LIN {X 0,Y 524.833,Z 335.716,A -85,B 0,C 180,E1 -4782.371,E2 -4782.371} C_VEL
LIN {X 0,Y 525.078,Z 323.315,A -85,B 0,C 180,E1 -4782.955,E2 -4782.955} C_VEL
LIN {X 0,Y 525.315,Z 310.12,A -85,B 0,C 180,E1 -4783.392,E2 -4783.392} C_VEL
LIN {X 0,Y 525.496,Z 297.421,A -85,B 0,C 180,E1 -4783.658,E2 -4783.658} C_VEL
LIN {X 0,Y 525.833,Z 204.394,A -85,B 0,C 180,E1 -4784.955,E2 -4784.955} C_VEL
LIN {X 0,Y 524.222,Z 193.612,A -85,B 0,C 180,E1 -4785.172,E2 -4785.172} C_VEL
LIN {X 0,Y 524.567,Z 175.695,A -85,B 0,C 180,E1 -4787.966,E2 -4787.966} C_VEL
LIN {X 0,Y 525.031,Z 156.558,A -85,B 0,C 180,E1 -4790.981,E2 -4790.981} C_VEL
LIN {X 0,Y 525.12,Z 144.956,A -85,B 0,C 180,E1 -4792.837,E2 -4792.837} C_VEL
LIN {X 0,Y 523.906,Z 138.227,A -85,B 0,C 180,E1 -4794.007,E2 -4794.007} C_VEL
LIN {X 0,Y 523.89,Z 138.23,A -85,B 0,C 180,E1 -4797.136,E2 -4797.136} C_VEL
LIN {X 0,Y 523.864,Z 138.233,A -85,B 0,C 180,E1 -4799.76,E2 -4799.76} C_VEL
LIN {X 0,Y 523.897,Z 138.225,A -85,B 0,C 180,E1 -4802.451,E2 -4802.451} C_VEL
LIN {X 0,Y 523.903,Z 138.229,A -85,B 0,C 180,E1 -4805.227,E2 -4805.227} C_VEL
LIN {X 0,Y 523.895,Z 138.223,A -85,B 0,C 180,E1 -4808.103,E2 -4808.103} C_VEL
LIN {X 0,Y 523.908,Z 138.227,A -85,B 0,C 180,E1 -4811.304,E2 -4811.304} C_VEL
LIN {X 0,Y 523.93,Z 138.224,A -85,B 0,C 180,E1 -4814.688,E2 -4814.688} C_VEL
LIN {X 0,Y 523.886,Z 138.222,A -85,B 0,C 180,E1 -4817.874,E2 -4817.874} C_VEL
LIN {X 0,Y 523.898,Z 138.229,A -85,B 0,C 180,E1 -4820.913,E2 -4820.913} C_VEL
LIN {X 0,Y 523.857,Z 138.225,A -85,B 0,C 180,E1 -4823.821,E2 -4823.821} C_VEL
LIN {X 0,Y 523.906,Z 138.226,A -85,B 0,C 180,E1 -4826.633,E2 -4826.633} C_VEL
LIN {X 0,Y 523.9,Z 138.22,A -85,B 0,C 180,E1 -4829.352,E2 -4829.352} C_VEL
LIN {X 0,Y 523.904,Z 138.225,A -85,B 0,C 180,E1 -4832.295,E2 -4832.295} C_VEL
LIN {X 0,Y 523.894,Z 138.222,A -85,B 0,C 180,E1 -4835.426,E2 -4835.426} C_VEL
LIN {X 0,Y 523.912,Z 138.219,A -85,B 0,C 180,E1 -4837.938,E2 -4837.938} C_VEL
LIN {X 0,Y 523.918,Z 138.225,A -85,B 0,C 180,E1 -4840.405,E2 -4840.405} C_VEL
LIN {X 0,Y 523.911,Z 138.222,A -85,B 0,C 180,E1 -4842.835,E2 -4842.835} C_VEL
LIN {X 0,Y 523.953,Z 138.213,A -85,B 0,C 180,E1 -4845.235,E2 -4845.235} C_VEL
LIN {X 0,Y 523.951,Z 138.22,A -85,B 0,C 180,E1 -4848.392,E2 -4848.392} C_VEL
LIN {X 0,Y 523.937,Z 138.217,A -85,B 0,C 180,E1 -4851.515,E2 -4851.515} C_VEL
LIN {X 0,Y 524.02,Z 138.206,A -85,B 0,C 180,E1 -4854.613,E2 -4854.613} C_VEL
LIN {X 0,Y 524.096,Z 138.202,A -85,B 0,C 180,E1 -4857.694,E2 -4857.694} C_VEL
LIN {X 0,Y 524.088,Z 138.205,A -85,B 0,C 180,E1 -4860,E2 -4860} C_VEL
LIN {X 0,Y 524.095,Z 138.2,A -85,B 0,C 180,E1 -4862.305,E2 -4862.305} C_VEL
LIN {X 0,Y 523.992,Z 138.214,A -85,B 0,C 180,E1 -4866.159,E2 -4866.159} C_VEL
LIN {X 0,Y 523.936,Z 138.221,A -85,B 0,C 180,E1 -4869.263,E2 -4869.263} C_VEL
LIN {X 0,Y 523.936,Z 138.22,A -85,B 0,C 180,E1 -4872.393,E2 -4872.393} C_VEL
LIN {X 0,Y 523.901,Z 138.231,A -85,B 0,C 180,E1 -4875.562,E2 -4875.562} C_VEL
LIN {X 0,Y 523.915,Z 138.221,A -85,B 0,C 180,E1 -4878.78,E2 -4878.78} C_VEL
LIN {X 0,Y 523.913,Z 138.227,A -85,B 0,C 180,E1 -4881.234,E2 -4881.234} C_VEL
LIN {X 0,Y 523.955,Z 138.316,A -85,B 0,C 180,E1 -4883.702,E2 -4883.702} C_VEL
LIN {X 0,Y 524.545,Z 142.807,A -85,B 0,C 180,E1 -4884.541,E2 -4884.541} C_VEL
LIN {X 0,Y 524.355,Z 157.183,A -85,B 0,C 180,E1 -4887.11,E2 -4887.11} C_VEL
LIN {X 0,Y 524.273,Z 167.066,A -85,B 0,C 180,E1 -4888.896,E2 -4888.896} C_VEL
LIN {X 0,Y 526.014,Z 177.203,A -85,B 0,C 180,E1 -4889.102,E2 -4889.102} C_VEL
LIN {X 0,Y 525.462,Z 274.648,A -85,B 0,C 180,E1 -4890.477,E2 -4890.477} C_VEL
LIN {X 0,Y 525.278,Z 287.649,A -85,B 0,C 180,E1 -4890.817,E2 -4890.817} C_VEL
LIN {X 0,Y 525.102,Z 299.989,A -85,B 0,C 180,E1 -4891.293,E2 -4891.293} C_VEL
LIN {X 0,Y 524.906,Z 309.383,A -85,B 0,C 180,E1 -4891.77,E2 -4891.77} C_VEL
LIN {X 0,Y 524.16,Z 314.614,A -85,B 0,C 180,E1 -4892.061,E2 -4892.061} C_VEL
LIN {X 0,Y 521.076,Z 322.898,A -85,B 0,C 180,E1 -4892.559,E2 -4892.559} C_VEL
LIN {X 0,Y 517.989,Z 330.723,A -85,B 0,C 180,E1 -4893.137,E2 -4893.137} C_VEL
LIN {X 0,Y 517.24,Z 335.226,A -85,B 0,C 180,E1 -4893.55,E2 -4893.55} C_VEL
LIN {X 0,Y 516.94,Z 344.855,A -85,B 0,C 180,E1 -4894.603,E2 -4894.603} C_VEL
LIN {X 0,Y 516.707,Z 353.618,A -85,B 0,C 180,E1 -4895.793,E2 -4895.793} C_VEL
LIN {X 0,Y 516.51,Z 360.825,A -85,B 0,C 180,E1 -4897.02,E2 -4897.02} C_VEL
LIN {X 0,Y 516.44,Z 366.704,A -85,B 0,C 180,E1 -4898.29,E2 -4898.29} C_VEL
LIN {X 0,Y 516.325,Z 370.782,A -85,B 0,C 180,E1 -4899.42,E2 -4899.42} C_VEL
LIN {X 0,Y 516.282,Z 374.444,A -85,B 0,C 180,E1 -4900.799,E2 -4900.799} C_VEL
LIN {X 0,Y 516.213,Z 376.306,A -85,B 0,C 180,E1 -4901.844,E2 -4901.844} C_VEL
LIN {X 0,Y 516.185,Z 377.467,A -85,B 0,C 180,E1 -4902.903,E2 -4902.903} C_VEL
LIN {X 0,Y 516.194,Z 377.886,A -85,B 0,C 180,E1 -4903.976,E2 -4903.976} C_VEL
LIN {X 0,Y 516.243,Z 377.53,A -85,B 0,C 180,E1 -4905.065,E2 -4905.065} C_VEL
LIN {X 0,Y 516.199,Z 376.374,A -85,B 0,C 180,E1 -4906.185,E2 -4906.185} C_VEL
LIN {X 0,Y 516.272,Z 373.361,A -85,B 0,C 180,E1 -4907.745,E2 -4907.745} C_VEL
LIN {X 0,Y 516.343,Z 370.205,A -85,B 0,C 180,E1 -4908.84,E2 -4908.84} C_VEL
LIN {X 0,Y 516.438,Z 364.785,A -85,B 0,C 180,E1 -4910.239,E2 -4910.239} C_VEL
LIN {X 0,Y 516.611,Z 358.52,A -85,B 0,C 180,E1 -4911.483,E2 -4911.483} C_VEL
LIN {X 0,Y 516.789,Z 350.403,A -85,B 0,C 180,E1 -4912.76,E2 -4912.76} C_VEL
LIN {X 0,Y 517.042,Z 341.469,A -85,B 0,C 180,E1 -4913.873,E2 -4913.873} C_VEL
LIN {X 0,Y 517.345,Z 331.353,A -85,B 0,C 180,E1 -4914.895,E2 -4914.895} C_VEL
LIN {X 0,Y 517.662,Z 320.358,A -85,B 0,C 180,E1 -4915.787,E2 -4915.787} C_VEL
LIN {X 0,Y 517.936,Z 308.363,A -85,B 0,C 180,E1 -4916.548,E2 -4916.548} C_VEL
LIN {X 0,Y 518.223,Z 297.272,A -85,B 0,C 180,E1 -4917.091,E2 -4917.091} C_VEL
LIN {X 0,Y 518.402,Z 284.135,A -85,B 0,C 180,E1 -4917.565,E2 -4917.565} C_VEL
LIN {X 0,Y 518.581,Z 270.861,A -85,B 0,C 180,E1 -4917.865,E2 -4917.865} C_VEL
LIN {X 0,Y 519.017,Z 176.794,A -85,B 0,C 180,E1 -4919.202,E2 -4919.202} C_VEL
LIN {X 0,Y 517.248,Z 167.254,A -85,B 0,C 180,E1 -4919.397,E2 -4919.397} C_VEL
LIN {X 0,Y 517.574,Z 152.214,A -85,B 0,C 180,E1 -4922.24,E2 -4922.24} C_VEL
LIN {X 0,Y 517.649,Z 143.381,A -85,B 0,C 180,E1 -4923.934,E2 -4923.934} C_VEL
LIN {X 0,Y 516.888,Z 139.103,A -85,B 0,C 180,E1 -4924.802,E2 -4924.802} C_VEL
LIN {X 0,Y 516.865,Z 139.099,A -85,B 0,C 180,E1 -4927.622,E2 -4927.622} C_VEL
LIN {X 0,Y 516.909,Z 139.096,A -85,B 0,C 180,E1 -4930.129,E2 -4930.129} C_VEL
LIN {X 0,Y 516.874,Z 139.103,A -85,B 0,C 180,E1 -4932.595,E2 -4932.595} C_VEL
LIN {X 0,Y 516.928,Z 139.091,A -85,B 0,C 180,E1 -4935.03,E2 -4935.03} C_VEL
LIN {X 0,Y 516.921,Z 139.097,A -85,B 0,C 180,E1 -4938.233,E2 -4938.233} C_VEL
LIN {X 0,Y 516.915,Z 139.091,A -85,B 0,C 180,E1 -4941.399,E2 -4941.399} C_VEL
LIN {X 0,Y 516.976,Z 139.087,A -85,B 0,C 180,E1 -4944.54,E2 -4944.54} C_VEL
LIN {X 0,Y 517.069,Z 139.074,A -85,B 0,C 180,E1 -4947.663,E2 -4947.663} C_VEL
LIN {X 0,Y 517.061,Z 139.08,A -85,B 0,C 180,E1 -4950,E2 -4950} C_VEL
LIN {X 0,Y 517.069,Z 139.076,A -85,B 0,C 180,E1 -4952.337,E2 -4952.337} C_VEL
LIN {X 0,Y 516.964,Z 139.089,A -85,B 0,C 180,E1 -4956.244,E2 -4956.244} C_VEL
LIN {X 0,Y 516.903,Z 139.095,A -85,B 0,C 180,E1 -4959.39,E2 -4959.39} C_VEL
LIN {X 0,Y 516.893,Z 139.094,A -85,B 0,C 180,E1 -4962.565,E2 -4962.565} C_VEL
LIN {X 0,Y 516.932,Z 139.09,A -85,B 0,C 180,E1 -4965.142,E2 -4965.142} C_VEL
LIN {X 0,Y 516.865,Z 139.099,A -85,B 0,C 180,E1 -4968.224,E2 -4968.224} C_VEL
LIN {X 0,Y 516.866,Z 139.097,A -85,B 0,C 180,E1 -4970.703,E2 -4970.703} C_VEL
LIN {X 0,Y 516.835,Z 139.105,A -85,B 0,C 180,E1 -4973.225,E2 -4973.225} C_VEL
LIN {X 0,Y 516.874,Z 139.097,A -85,B 0,C 180,E1 -4976.181,E2 -4976.181} C_VEL
LIN {X 0,Y 516.824,Z 139.102,A -85,B 0,C 180,E1 -4978.421,E2 -4978.421} C_VEL
LIN {X 0,Y 516.872,Z 139.101,A -85,B 0,C 180,E1 -4981.11,E2 -4981.11} C_VEL
LIN {X 0,Y 516.875,Z 139.097,A -85,B 0,C 180,E1 -4983.961,E2 -4983.961} C_VEL
LIN {X 0,Y 516.843,Z 139.102,A -85,B 0,C 180,E1 -4986.748,E2 -4986.748} C_VEL
LIN {X 0,Y 516.852,Z 139.101,A -85,B 0,C 180,E1 -4989.724,E2 -4989.724} C_VEL
LIN {X 0,Y 516.835,Z 139.105,A -85,B 0,C 180,E1 -4992.836,E2 -4992.836} C_VEL
LIN {X 0,Y 516.89,Z 139.102,A -85,B 0,C 180,E1 -4995.007,E2 -4995.007} C_VEL
LIN {X 0,Y 516.846,Z 139.101,A -85,B 0,C 180,E1 -4998.406,E2 -4998.406} C_VEL
LIN {X 0,Y 516.866,Z 139.101,A -85,B 0,C 180,E1 -5001.283,E2 -5001.283} C_VEL
LIN {X 0,Y 516.844,Z 139.106,A -85,B 0,C 180,E1 -5004.673,E2 -5004.673} C_VEL
LIN {X 0,Y 516.885,Z 139.096,A -85,B 0,C 180,E1 -5007.458,E2 -5007.458} C_VEL
LIN {X 0,Y 516.89,Z 139.103,A -85,B 0,C 180,E1 -5010.694,E2 -5010.694} C_VEL
LIN {X 0,Y 516.872,Z 139.096,A -85,B 0,C 180,E1 -5013.819,E2 -5013.819} C_VEL
LIN {X 0,Y 516.834,Z 139.107,A -85,B 0,C 180,E1 -5016.775,E2 -5016.775} C_VEL
LIN {X 0,Y 516.899,Z 139.093,A -85,B 0,C 180,E1 -5019.742,E2 -5019.742} C_VEL
LIN {X 0,Y 516.871,Z 139.103,A -85,B 0,C 180,E1 -5022.595,E2 -5022.595} C_VEL
LIN {X 0,Y 516.925,Z 139.091,A -85,B 0,C 180,E1 -5025.03,E2 -5025.03} C_VEL
LIN {X 0,Y 516.918,Z 139.098,A -85,B 0,C 180,E1 -5028.233,E2 -5028.233} C_VEL
LIN {X 0,Y 516.912,Z 139.091,A -85,B 0,C 180,E1 -5031.399,E2 -5031.399} C_VEL
LIN {X 0,Y 516.973,Z 139.087,A -85,B 0,C 180,E1 -5034.54,E2 -5034.54} C_VEL
LIN {X 0,Y 517.066,Z 139.075,A -85,B 0,C 180,E1 -5037.663,E2 -5037.663} C_VEL
LIN {X 0,Y 517.058,Z 139.081,A -85,B 0,C 180,E1 -5040,E2 -5040} C_VEL
LIN {X 0,Y 517.066,Z 139.076,A -85,B 0,C 180,E1 -5042.337,E2 -5042.337} C_VEL
LIN {X 0,Y 516.961,Z 139.089,A -85,B 0,C 180,E1 -5046.244,E2 -5046.244} C_VEL
LIN {X 0,Y 516.9,Z 139.095,A -85,B 0,C 180,E1 -5049.391,E2 -5049.391} C_VEL
LIN {X 0,Y 516.89,Z 139.094,A -85,B 0,C 180,E1 -5052.565,E2 -5052.565} C_VEL
LIN {X 0,Y 516.93,Z 139.091,A -85,B 0,C 180,E1 -5055.142,E2 -5055.142} C_VEL
LIN {X 0,Y 516.864,Z 139.099,A -85,B 0,C 180,E1 -5058.225,E2 -5058.225} C_VEL
LIN {X 0,Y 516.865,Z 139.097,A -85,B 0,C 180,E1 -5060.704,E2 -5060.704} C_VEL
LIN {X 0,Y 516.834,Z 139.105,A -85,B 0,C 180,E1 -5063.226,E2 -5063.226} C_VEL
LIN {X 0,Y 516.874,Z 139.097,A -85,B 0,C 180,E1 -5066.182,E2 -5066.182} C_VEL
LIN {X 0,Y 516.824,Z 139.102,A -85,B 0,C 180,E1 -5068.421,E2 -5068.421} C_VEL
LIN {X 0,Y 516.844,Z 139.105,A -85,B 0,C 180,E1 -5071.113,E2 -5071.113} C_VEL
LIN {X 0,Y 516.876,Z 139.097,A -85,B 0,C 180,E1 -5073.962,E2 -5073.962} C_VEL
LIN {X 0,Y 516.811,Z 139.106,A -85,B 0,C 180,E1 -5076.752,E2 -5076.752} C_VEL
LIN {X 0,Y 516.853,Z 139.1,A -85,B 0,C 180,E1 -5079.724,E2 -5079.724} C_VEL
LIN {X 0,Y 516.838,Z 139.105,A -85,B 0,C 180,E1 -5082.837,E2 -5082.837} C_VEL
LIN {X 0,Y 516.894,Z 139.102,A -85,B 0,C 180,E1 -5085.007,E2 -5085.007} C_VEL
LIN {X 0,Y 516.847,Z 139.101,A -85,B 0,C 180,E1 -5088.408,E2 -5088.408} C_VEL
LIN {X 0,Y 516.867,Z 139.1,A -85,B 0,C 180,E1 -5091.283,E2 -5091.283} C_VEL
LIN {X 0,Y 516.847,Z 139.106,A -85,B 0,C 180,E1 -5094.674,E2 -5094.674} C_VEL
LIN {X 0,Y 516.866,Z 139.098,A -85,B 0,C 180,E1 -5097.462,E2 -5097.462} C_VEL
LIN {X 0,Y 516.837,Z 139.107,A -85,B 0,C 180,E1 -5100.491,E2 -5100.491} C_VEL
LIN {X 0,Y 516.828,Z 139.103,A -85,B 0,C 180,E1 -5103.337,E2 -5103.337} C_VEL
LIN {X 0,Y 516.857,Z 139.147,A -85,B 0,C 180,E1 -5105.691,E2 -5105.691} C_VEL
LIN {X 0,Y 518.326,Z 147.13,A -85,B 0,C 180,E1 -5107.091,E2 -5107.091} C_VEL
LIN {X 0,Y 518.015,Z 161.935,A -85,B 0,C 180,E1 -5109.52,E2 -5109.52} C_VEL
LIN {X 0,Y 517.575,Z 178.892,A -85,B 0,C 180,E1 -5112.257,E2 -5112.257} C_VEL
LIN {X 0,Y 517.266,Z 193.985,A -85,B 0,C 180,E1 -5114.641,E2 -5114.641} C_VEL
LIN {X 0,Y 519.025,Z 206.11,A -85,B 0,C 180,E1 -5114.869,E2 -5114.869} C_VEL
LIN {X 0,Y 518.545,Z 302.791,A -85,B 0,C 180,E1 -5116.255,E2 -5116.255} C_VEL
LIN {X 0,Y 518.28,Z 316.493,A -85,B 0,C 180,E1 -5116.622,E2 -5116.622} C_VEL
LIN {X 0,Y 518.045,Z 328.834,A -85,B 0,C 180,E1 -5117.115,E2 -5117.115} C_VEL
LIN {X 0,Y 517.691,Z 341.583,A -85,B 0,C 180,E1 -5117.81,E2 -5117.81} C_VEL
LIN {X 0,Y 517.429,Z 353.383,A -85,B 0,C 180,E1 -5118.642,E2 -5118.642} C_VEL
LIN {X 0,Y 517.158,Z 362.386,A -85,B 0,C 180,E1 -5119.429,E2 -5119.429} C_VEL
LIN {X 0,Y 516.9,Z 371.625,A -85,B 0,C 180,E1 -5120.412,E2 -5120.412} C_VEL
LIN {X 0,Y 516.652,Z 380.613,A -85,B 0,C 180,E1 -5121.591,E2 -5121.591} C_VEL
LIN {X 0,Y 516.503,Z 387.85,A -85,B 0,C 180,E1 -5122.769,E2 -5122.769} C_VEL
LIN {X 0,Y 516.385,Z 392.73,A -85,B 0,C 180,E1 -5123.749,E2 -5123.749} C_VEL
LIN {X 0,Y 516.312,Z 397.472,A -85,B 0,C 180,E1 -5124.924,E2 -5124.924} C_VEL
LIN {X 0,Y 516.352,Z 401.097,A -85,B 0,C 180,E1 -5126.098,E2 -5126.098} C_VEL
LIN {X 0,Y 516.283,Z 402.964,A -85,B 0,C 180,E1 -5126.879,E2 -5126.879} C_VEL
LIN {X 0,Y 516.261,Z 404.365,A -85,B 0,C 180,E1 -5127.659,E2 -5127.659} C_VEL
LIN {X 0,Y 516.162,Z 405.968,A -85,B 0,C 180,E1 -5129.22,E2 -5129.22} C_VEL
LIN {X 0,Y 516.159,Z 406.183,A -85,B 0,C 180,E1 -5130,E2 -5130} C_VEL
LIN {X 0,Y 516.192,Z 405.353,A -85,B 0,C 180,E1 -5131.56,E2 -5131.56} C_VEL
LIN {X 0,Y 516.261,Z 404.351,A -85,B 0,C 180,E1 -5132.34,E2 -5132.34} C_VEL
LIN {X 0,Y 516.282,Z 402.945,A -85,B 0,C 180,E1 -5133.121,E2 -5133.121} C_VEL
LIN {X 0,Y 516.31,Z 399.992,A -85,B 0,C 180,E1 -5134.293,E2 -5134.293} C_VEL
LIN {X 0,Y 516.368,Z 395.995,A -85,B 0,C 180,E1 -5135.467,E2 -5135.467} C_VEL
LIN {X 0,Y 516.44,Z 390.084,A -85,B 0,C 180,E1 -5136.792,E2 -5136.792} C_VEL
LIN {X 0,Y 516.586,Z 383.121,A -85,B 0,C 180,E1 -5138.016,E2 -5138.016} C_VEL
LIN {X 0,Y 516.772,Z 374.778,A -85,B 0,C 180,E1 -5139.195,E2 -5139.195} C_VEL
LIN {X 0,Y 516.997,Z 366.207,A -85,B 0,C 180,E1 -5140.179,E2 -5140.179} C_VEL
LIN {X 0,Y 517.317,Z 355.623,A -85,B 0,C 180,E1 -5141.162,E2 -5141.162} C_VEL
LIN {X 0,Y 517.608,Z 344.508,A -85,B 0,C 180,E1 -5141.994,E2 -5141.994} C_VEL
LIN {X 0,Y 517.939,Z 333.614,A -85,B 0,C 180,E1 -5142.638,E2 -5142.638} C_VEL
LIN {X 0,Y 518.168,Z 321.669,A -85,B 0,C 180,E1 -5143.181,E2 -5143.181} C_VEL
LIN {X 0,Y 518.445,Z 307.88,A -85,B 0,C 180,E1 -5143.623,E2 -5143.623} C_VEL
LIN {X 0,Y 518.626,Z 295.308,A -85,B 0,C 180,E1 -5143.868,E2 -5143.868} C_VEL
LIN {X 0,Y 518.957,Z 204.938,A -85,B 0,C 180,E1 -5145.147,E2 -5145.147} C_VEL
LIN {X 0,Y 517.222,Z 193.364,A -85,B 0,C 180,E1 -5145.387,E2 -5145.387} C_VEL
LIN {X 0,Y 517.665,Z 174.314,A -85,B 0,C 180,E1 -5148.4,E2 -5148.4} C_VEL
LIN {X 0,Y 518.083,Z 155.034,A -85,B 0,C 180,E1 -5151.485,E2 -5151.485} C_VEL
LIN {X 0,Y 518.193,Z 146.314,A -85,B 0,C 180,E1 -5152.899,E2 -5152.899} C_VEL
LIN {X 0,Y 516.869,Z 139.103,A -85,B 0,C 180,E1 -5154.169,E2 -5154.169} C_VEL
LIN {X 0,Y 516.827,Z 139.107,A -85,B 0,C 180,E1 -5156.663,E2 -5156.663} C_VEL
LIN {X 0,Y 516.836,Z 139.112,A -85,B 0,C 180,E1 -5159.508,E2 -5159.508} C_VEL
LIN {X 0,Y 516.865,Z 139.101,A -85,B 0,C 180,E1 -5162.537,E2 -5162.537} C_VEL
LIN {X 0,Y 516.846,Z 139.108,A -85,B 0,C 180,E1 -5165.326,E2 -5165.326} C_VEL
LIN {X 0,Y 516.865,Z 139.103,A -85,B 0,C 180,E1 -5168.716,E2 -5168.716} C_VEL
LIN {X 0,Y 516.841,Z 139.103,A -85,B 0,C 180,E1 -5171.781,E2 -5171.781} C_VEL
LIN {X 0,Y 516.892,Z 139.102,A -85,B 0,C 180,E1 -5175.006,E2 -5175.006} C_VEL
LIN {X 0,Y 516.843,Z 139.102,A -85,B 0,C 180,E1 -5178.406,E2 -5178.406} C_VEL
LIN {X 0,Y 516.864,Z 139.101,A -85,B 0,C 180,E1 -5181.282,E2 -5181.282} C_VEL
LIN {X 0,Y 516.845,Z 139.107,A -85,B 0,C 180,E1 -5184.672,E2 -5184.672} C_VEL
LIN {X 0,Y 516.886,Z 139.095,A -85,B 0,C 180,E1 -5187.457,E2 -5187.457} C_VEL
LIN {X 0,Y 516.819,Z 139.11,A -85,B 0,C 180,E1 -5190.689,E2 -5190.689} C_VEL
LIN {X 0,Y 516.83,Z 139.1,A -85,B 0,C 180,E1 -5193.337,E2 -5193.337} C_VEL
LIN {X 0,Y 516.873,Z 139.098,A -85,B 0,C 180,E1 -5195.926,E2 -5195.926} C_VEL
LIN {X 0,Y 516.845,Z 139.107,A -85,B 0,C 180,E1 -5198.46,E2 -5198.46} C_VEL
LIN {X 0,Y 516.856,Z 139.098,A -85,B 0,C 180,E1 -5200.953,E2 -5200.953} C_VEL
LIN {X 0,Y 516.832,Z 139.102,A -85,B 0,C 180,E1 -5203.407,E2 -5203.407} C_VEL
LIN {X 0,Y 516.861,Z 139.099,A -85,B 0,C 180,E1 -5205.832,E2 -5205.832} C_VEL
LIN {X 0,Y 516.917,Z 139.097,A -85,B 0,C 180,E1 -5208.232,E2 -5208.232} C_VEL
LIN {X 0,Y 516.911,Z 139.092,A -85,B 0,C 180,E1 -5211.398,E2 -5211.398} C_VEL
LIN {X 0,Y 516.971,Z 139.085,A -85,B 0,C 180,E1 -5214.539,E2 -5214.539} C_VEL
LIN {X 0,Y 517.065,Z 139.077,A -85,B 0,C 180,E1 -5217.663,E2 -5217.663} C_VEL
LIN {X 0,Y 517.056,Z 139.081,A -85,B 0,C 180,E1 -5220,E2 -5220} C_VEL
LIN {X 0,Y 517.064,Z 139.076,A -85,B 0,C 180,E1 -5222.337,E2 -5222.337} C_VEL
LIN {X 0,Y 516.959,Z 139.09,A -85,B 0,C 180,E1 -5226.243,E2 -5226.243} C_VEL
LIN {X 0,Y 516.898,Z 139.099,A -85,B 0,C 180,E1 -5229.39,E2 -5229.39} C_VEL
LIN {X 0,Y 516.888,Z 139.098,A -85,B 0,C 180,E1 -5232.565,E2 -5232.565} C_VEL
LIN {X 0,Y 516.927,Z 139.096,A -85,B 0,C 180,E1 -5235.142,E2 -5235.142} C_VEL
LIN {X 0,Y 516.864,Z 139.1,A -85,B 0,C 180,E1 -5238.224,E2 -5238.224} C_VEL
LIN {X 0,Y 516.881,Z 139.099,A -85,B 0,C 180,E1 -5240.702,E2 -5240.702} C_VEL
LIN {X 0,Y 516.916,Z 139.208,A -85,B 0,C 180,E1 -5243.566,E2 -5243.566} C_VEL
LIN {X 0,Y 517.58,Z 144.348,A -85,B 0,C 180,E1 -5244.529,E2 -5244.529} C_VEL
LIN {X 0,Y 517.381,Z 159.561,A -85,B 0,C 180,E1 -5247.287,E2 -5247.287} C_VEL
LIN {X 0,Y 517.289,Z 167.305,A -85,B 0,C 180,E1 -5248.697,E2 -5248.697} C_VEL
LIN {X 0,Y 519.071,Z 177.126,A -85,B 0,C 180,E1 -5248.894,E2 -5248.894} C_VEL
LIN {X 0,Y 518.568,Z 275.171,A -85,B 0,C 180,E1 -5250.306,E2 -5250.306} C_VEL
LIN {X 0,Y 518.367,Z 288.716,A -85,B 0,C 180,E1 -5250.671,E2 -5250.671} C_VEL
LIN {X 0,Y 518.18,Z 299.936,A -85,B 0,C 180,E1 -5251.114,E2 -5251.114} C_VEL
LIN {X 0,Y 517.874,Z 312.383,A -85,B 0,C 180,E1 -5251.772,E2 -5251.772} C_VEL
LIN {X 0,Y 517.567,Z 324.128,A -85,B 0,C 180,E1 -5252.582,E2 -5252.582} C_VEL
LIN {X 0,Y 517.245,Z 334.754,A -85,B 0,C 180,E1 -5253.503,E2 -5253.503} C_VEL
LIN {X 0,Y 517.24,Z 335.226,A -85,B 0,C 180,E1 -5253.55,E2 -5253.55} C_VEL
LIN {X 0,Y 516.498,Z 339.613,A -85,B 0,C 180,E1 -5253.989,E2 -5253.989} C_VEL
LIN {X 0,Y 513.417,Z 346.426,A -85,B 0,C 180,E1 -5254.721,E2 -5254.721} C_VEL
LIN {X 0,Y 510.347,Z 352.625,A -85,B 0,C 180,E1 -5255.514,E2 -5255.514} C_VEL
LIN {X 0,Y 509.621,Z 356.065,A -85,B 0,C 180,E1 -5256.042,E2 -5256.042} C_VEL
LIN {X 0,Y 509.438,Z 363.245,A -85,B 0,C 180,E1 -5257.373,E2 -5257.373} C_VEL
LIN {X 0,Y 509.344,Z 367.586,A -85,B 0,C 180,E1 -5258.383,E2 -5258.383} C_VEL
LIN {X 0,Y 509.223,Z 372.606,A -85,B 0,C 180,E1 -5259.923,E2 -5259.923} C_VEL
LIN {X 0,Y 509.196,Z 374.321,A -85,B 0,C 180,E1 -5260.615,E2 -5260.615} C_VEL
LIN {X 0,Y 509.117,Z 376.485,A -85,B 0,C 180,E1 -5261.805,E2 -5261.805} C_VEL
LIN {X 0,Y 509.097,Z 377.713,A -85,B 0,C 180,E1 -5262.976,E2 -5262.976} C_VEL
LIN {X 0,Y 509.11,Z 378.078,A -85,B 0,C 180,E1 -5264.125,E2 -5264.125} C_VEL
LIN {X 0,Y 509.142,Z 377.615,A -85,B 0,C 180,E1 -5265.253,E2 -5265.253} C_VEL
LIN {X 0,Y 509.108,Z 376.365,A -85,B 0,C 180,E1 -5266.353,E2 -5266.353} C_VEL
LIN {X 0,Y 509.145,Z 374.368,A -85,B 0,C 180,E1 -5267.44,E2 -5267.44} C_VEL
LIN {X 0,Y 509.272,Z 370.168,A -85,B 0,C 180,E1 -5268.975,E2 -5268.975} C_VEL
LIN {X 0,Y 509.371,Z 364.864,A -85,B 0,C 180,E1 -5270.349,E2 -5270.349} C_VEL
LIN {X 0,Y 509.569,Z 358.394,A -85,B 0,C 180,E1 -5271.638,E2 -5271.638} C_VEL
LIN {X 0,Y 509.757,Z 350.41,A -85,B 0,C 180,E1 -5272.902,E2 -5272.902} C_VEL
LIN {X 0,Y 510.045,Z 341.308,A -85,B 0,C 180,E1 -5274.045,E2 -5274.045} C_VEL
LIN {X 0,Y 510.341,Z 331.71,A -85,B 0,C 180,E1 -5275.025,E2 -5275.025} C_VEL
LIN {X 0,Y 510.674,Z 321.298,A -85,B 0,C 180,E1 -5275.889,E2 -5275.889} C_VEL
LIN {X 0,Y 510.99,Z 309.187,A -85,B 0,C 180,E1 -5276.678,E2 -5276.678} C_VEL
LIN {X 0,Y 511.308,Z 296.926,A -85,B 0,C 180,E1 -5277.289,E2 -5277.289} C_VEL
LIN {X 0,Y 511.518,Z 283.934,A -85,B 0,C 180,E1 -5277.756,E2 -5277.756} C_VEL
LIN {X 0,Y 511.714,Z 270.642,A -85,B 0,C 180,E1 -5278.056,E2 -5278.056} C_VEL
LIN {X 0,Y 512.281,Z 178.46,A -85,B 0,C 180,E1 -5279.382,E2 -5279.382} C_VEL
LIN {X 0,Y 510.264,Z 167.381,A -85,B 0,C 180,E1 -5279.617,E2 -5279.617} C_VEL
LIN {X 0,Y 510.608,Z 152.103,A -85,B 0,C 180,E1 -5282.543,E2 -5282.543} C_VEL
LIN {X 0,Y 510.729,Z 145.206,A -85,B 0,C 180,E1 -5283.875,E2 -5283.875} C_VEL
LIN {X 0,Y 509.845,Z 139.98,A -85,B 0,C 180,E1 -5284.974,E2 -5284.974} C_VEL
LIN {X 0,Y 509.804,Z 139.982,A -85,B 0,C 180,E1 -5288.148,E2 -5288.148} C_VEL
LIN {X 0,Y 509.839,Z 139.98,A -85,B 0,C 180,E1 -5290.681,E2 -5290.681} C_VEL
LIN {X 0,Y 509.791,Z 139.979,A -85,B 0,C 180,E1 -5293.172,E2 -5293.172} C_VEL
LIN {X 0,Y 509.84,Z 139.973,A -85,B 0,C 180,E1 -5295.634,E2 -5295.634} C_VEL
LIN {X 0,Y 509.885,Z 139.972,A -85,B 0,C 180,E1 -5298.131,E2 -5298.131} C_VEL
LIN {X 0,Y 509.868,Z 139.969,A -85,B 0,C 180,E1 -5301.279,E2 -5301.279} C_VEL
LIN {X 0,Y 509.912,Z 139.965,A -85,B 0,C 180,E1 -5303.67,E2 -5303.67} C_VEL
LIN {X 0,Y 509.881,Z 139.968,A -85,B 0,C 180,E1 -5306.84,E2 -5306.84} C_VEL
LIN {X 0,Y 509.919,Z 139.967,A -85,B 0,C 180,E1 -5308.421,E2 -5308.421} C_VEL
LIN {X 0,Y 510.03,Z 139.956,A -85,B 0,C 180,E1 -5310,E2 -5310} C_VEL
LIN {X 0,Y 510.038,Z 139.952,A -85,B 0,C 180,E1 -5312.369,E2 -5312.369} C_VEL
LIN {X 0,Y 509.931,Z 139.964,A -85,B 0,C 180,E1 -5315.536,E2 -5315.536} C_VEL
LIN {X 0,Y 509.871,Z 139.977,A -85,B 0,C 180,E1 -5317.923,E2 -5317.923} C_VEL
LIN {X 0,Y 509.858,Z 139.971,A -85,B 0,C 180,E1 -5321.127,E2 -5321.127} C_VEL
LIN {X 0,Y 509.82,Z 139.98,A -85,B 0,C 180,E1 -5323.553,E2 -5323.553} C_VEL
LIN {X 0,Y 509.798,Z 139.982,A -85,B 0,C 180,E1 -5326.005,E2 -5326.005} C_VEL
LIN {X 0,Y 509.822,Z 139.975,A -85,B 0,C 180,E1 -5328.485,E2 -5328.485} C_VEL
LIN {X 0,Y 509.813,Z 139.977,A -85,B 0,C 180,E1 -5331.003,E2 -5331.003} C_VEL
LIN {X 0,Y 509.803,Z 139.986,A -85,B 0,C 180,E1 -5333.565,E2 -5333.565} C_VEL
LIN {X 0,Y 509.81,Z 139.976,A -85,B 0,C 180,E1 -5336.356,E2 -5336.356} C_VEL
LIN {X 0,Y 509.788,Z 139.98,A -85,B 0,C 180,E1 -5338.849,E2 -5338.849} C_VEL
LIN {X 0,Y 509.806,Z 139.982,A -85,B 0,C 180,E1 -5341.591,E2 -5341.591} C_VEL
LIN {X 0,Y 509.828,Z 139.974,A -85,B 0,C 180,E1 -5344.415,E2 -5344.415} C_VEL
LIN {X 0,Y 509.8,Z 139.985,A -85,B 0,C 180,E1 -5347.342,E2 -5347.342} C_VEL
LIN {X 0,Y 509.806,Z 139.977,A -85,B 0,C 180,E1 -5350.385,E2 -5350.385} C_VEL
LIN {X 0,Y 509.799,Z 139.98,A -85,B 0,C 180,E1 -5353.573,E2 -5353.573} C_VEL
LIN {X 0,Y 509.799,Z 139.979,A -85,B 0,C 180,E1 -5356.426,E2 -5356.426} C_VEL
LIN {X 0,Y 509.807,Z 139.977,A -85,B 0,C 180,E1 -5359.615,E2 -5359.615} C_VEL
LIN {X 0,Y 509.776,Z 139.985,A -85,B 0,C 180,E1 -5362.656,E2 -5362.656} C_VEL
LIN {X 0,Y 509.831,Z 139.973,A -85,B 0,C 180,E1 -5365.801,E2 -5365.801} C_VEL
LIN {X 0,Y 509.83,Z 139.982,A -85,B 0,C 180,E1 -5368.722,E2 -5368.722} C_VEL
LIN {X 0,Y 509.823,Z 139.977,A -85,B 0,C 180,E1 -5371.153,E2 -5371.153} C_VEL
LIN {X 0,Y 509.84,Z 139.972,A -85,B 0,C 180,E1 -5373.826,E2 -5373.826} C_VEL
LIN {X 0,Y 509.801,Z 139.983,A -85,B 0,C 180,E1 -5376.436,E2 -5376.436} C_VEL
LIN {X 0,Y 509.882,Z 139.968,A -85,B 0,C 180,E1 -5379.844,E2 -5379.844} C_VEL
LIN {X 0,Y 509.845,Z 139.979,A -85,B 0,C 180,E1 -5382.347,E2 -5382.347} C_VEL
LIN {X 0,Y 509.877,Z 139.971,A -85,B 0,C 180,E1 -5384.818,E2 -5384.818} C_VEL
LIN {X 0,Y 509.882,Z 139.973,A -85,B 0,C 180,E1 -5388.131,E2 -5388.131} C_VEL
LIN {X 0,Y 509.865,Z 139.969,A -85,B 0,C 180,E1 -5391.279,E2 -5391.279} C_VEL
LIN {X 0,Y 509.909,Z 139.965,A -85,B 0,C 180,E1 -5393.67,E2 -5393.67} C_VEL
LIN {X 0,Y 509.878,Z 139.968,A -85,B 0,C 180,E1 -5396.84,E2 -5396.84} C_VEL
LIN {X 0,Y 509.916,Z 139.967,A -85,B 0,C 180,E1 -5398.421,E2 -5398.421} C_VEL
LIN {X 0,Y 510.027,Z 139.957,A -85,B 0,C 180,E1 -5400,E2 -5400} C_VEL
LIN {X 0,Y 510.035,Z 139.952,A -85,B 0,C 180,E1 -5402.37,E2 -5402.37} C_VEL
LIN {X 0,Y 509.928,Z 139.964,A -85,B 0,C 180,E1 -5405.537,E2 -5405.537} C_VEL
LIN {X 0,Y 509.868,Z 139.977,A -85,B 0,C 180,E1 -5407.923,E2 -5407.923} C_VEL
LIN {X 0,Y 509.856,Z 139.971,A -85,B 0,C 180,E1 -5411.127,E2 -5411.127} C_VEL
LIN {X 0,Y 509.817,Z 139.981,A -85,B 0,C 180,E1 -5413.554,E2 -5413.554} C_VEL
LIN {X 0,Y 509.796,Z 139.982,A -85,B 0,C 180,E1 -5416.005,E2 -5416.005} C_VEL
LIN {X 0,Y 509.82,Z 139.975,A -85,B 0,C 180,E1 -5418.486,E2 -5418.486} C_VEL
LIN {X 0,Y 509.812,Z 139.977,A -85,B 0,C 180,E1 -5421.004,E2 -5421.004} C_VEL
LIN {X 0,Y 509.802,Z 139.985,A -85,B 0,C 180,E1 -5423.565,E2 -5423.565} C_VEL
LIN {X 0,Y 509.81,Z 139.976,A -85,B 0,C 180,E1 -5426.357,E2 -5426.357} C_VEL
LIN {X 0,Y 509.788,Z 139.98,A -85,B 0,C 180,E1 -5428.85,E2 -5428.85} C_VEL
LIN {X 0,Y 509.792,Z 139.983,A -85,B 0,C 180,E1 -5431.592,E2 -5431.592} C_VEL
LIN {X 0,Y 509.829,Z 139.974,A -85,B 0,C 180,E1 -5434.416,E2 -5434.416} C_VEL
LIN {X 0,Y 509.779,Z 139.987,A -85,B 0,C 180,E1 -5437.344,E2 -5437.344} C_VEL
LIN {X 0,Y 509.809,Z 139.976,A -85,B 0,C 180,E1 -5440.385,E2 -5440.385} C_VEL
LIN {X 0,Y 509.79,Z 139.981,A -85,B 0,C 180,E1 -5443.575,E2 -5443.575} C_VEL
LIN {X 0,Y 509.79,Z 139.98,A -85,B 0,C 180,E1 -5446.426,E2 -5446.426} C_VEL
LIN {X 0,Y 509.81,Z 139.977,A -85,B 0,C 180,E1 -5449.616,E2 -5449.616} C_VEL
LIN {X 0,Y 509.778,Z 139.985,A -85,B 0,C 180,E1 -5452.656,E2 -5452.656} C_VEL
LIN {X 0,Y 509.837,Z 139.972,A -85,B 0,C 180,E1 -5455.801,E2 -5455.801} C_VEL
LIN {X 0,Y 509.814,Z 139.984,A -85,B 0,C 180,E1 -5458.727,E2 -5458.727} C_VEL
LIN {X 0,Y 509.822,Z 139.977,A -85,B 0,C 180,E1 -5462.051,E2 -5462.051} C_VEL
LIN {X 0,Y 509.783,Z 139.984,A -85,B 0,C 180,E1 -5464.699,E2 -5464.699} C_VEL
LIN {X 0,Y 509.824,Z 140.059,A -85,B 0,C 180,E1 -5465.52,E2 -5465.52} C_VEL
LIN {X 0,Y 511.39,Z 148.609,A -85,B 0,C 180,E1 -5467.041,E2 -5467.041} C_VEL
LIN {X 0,Y 511.01,Z 163.768,A -85,B 0,C 180,E1 -5469.56,E2 -5469.56} C_VEL
LIN {X 0,Y 510.593,Z 179.025,A -85,B 0,C 180,E1 -5472.058,E2 -5472.058} C_VEL
LIN {X 0,Y 510.228,Z 193.618,A -85,B 0,C 180,E1 -5474.421,E2 -5474.421} C_VEL
LIN {X 0,Y 512.206,Z 207.217,A -85,B 0,C 180,E1 -5474.681,E2 -5474.681} C_VEL
LIN {X 0,Y 511.649,Z 302.381,A -85,B 0,C 180,E1 -5476.066,E2 -5476.066} C_VEL
LIN {X 0,Y 511.385,Z 316.153,A -85,B 0,C 180,E1 -5476.438,E2 -5476.438} C_VEL
LIN {X 0,Y 511.084,Z 328.539,A -85,B 0,C 180,E1 -5476.936,E2 -5476.936} C_VEL
LIN {X 0,Y 510.743,Z 341.132,A -85,B 0,C 180,E1 -5477.63,E2 -5477.63} C_VEL
LIN {X 0,Y 510.484,Z 351.842,A -85,B 0,C 180,E1 -5478.384,E2 -5478.384} C_VEL
LIN {X 0,Y 510.161,Z 362.147,A -85,B 0,C 180,E1 -5479.282,E2 -5479.282} C_VEL
LIN {X 0,Y 509.847,Z 371.396,A -85,B 0,C 180,E1 -5480.278,E2 -5480.278} C_VEL
LIN {X 0,Y 509.606,Z 380.394,A -85,B 0,C 180,E1 -5481.474,E2 -5481.474} C_VEL
LIN {X 0,Y 509.428,Z 387.637,A -85,B 0,C 180,E1 -5482.668,E2 -5482.668} C_VEL
LIN {X 0,Y 509.309,Z 392.523,A -85,B 0,C 180,E1 -5483.662,E2 -5483.662} C_VEL
LIN {X 0,Y 509.241,Z 397.271,A -85,B 0,C 180,E1 -5484.853,E2 -5484.853} C_VEL
LIN {X 0,Y 509.245,Z 400.899,A -85,B 0,C 180,E1 -5486.043,E2 -5486.043} C_VEL
LIN {X 0,Y 509.2,Z 402.769,A -85,B 0,C 180,E1 -5486.835,E2 -5486.835} C_VEL
LIN {X 0,Y 509.19,Z 404.17,A -85,B 0,C 180,E1 -5487.627,E2 -5487.627} C_VEL
LIN {X 0,Y 509.076,Z 405.774,A -85,B 0,C 180,E1 -5489.209,E2 -5489.209} C_VEL
LIN {X 0,Y 509.07,Z 405.989,A -85,B 0,C 180,E1 -5490,E2 -5490} C_VEL
LIN {X 0,Y 509.113,Z 405.156,A -85,B 0,C 180,E1 -5491.582,E2 -5491.582} C_VEL
LIN {X 0,Y 509.19,Z 404.153,A -85,B 0,C 180,E1 -5492.373,E2 -5492.373} C_VEL
LIN {X 0,Y 509.2,Z 402.744,A -85,B 0,C 180,E1 -5493.165,E2 -5493.165} C_VEL
LIN {X 0,Y 509.202,Z 399.786,A -85,B 0,C 180,E1 -5494.353,E2 -5494.353} C_VEL
LIN {X 0,Y 509.283,Z 395.783,A -85,B 0,C 180,E1 -5495.543,E2 -5495.543} C_VEL
LIN {X 0,Y 509.395,Z 389.723,A -85,B 0,C 180,E1 -5496.914,E2 -5496.914} C_VEL
LIN {X 0,Y 509.536,Z 382.889,A -85,B 0,C 180,E1 -5498.127,E2 -5498.127} C_VEL
LIN {X 0,Y 509.732,Z 374.535,A -85,B 0,C 180,E1 -5499.323,E2 -5499.323} C_VEL
LIN {X 0,Y 509.969,Z 365.95,A -85,B 0,C 180,E1 -5500.32,E2 -5500.32} C_VEL
LIN {X 0,Y 510.333,Z 355.35,A -85,B 0,C 180,E1 -5501.317,E2 -5501.317} C_VEL
LIN {X 0,Y 510.644,Z 344.218,A -85,B 0,C 180,E1 -5502.16,E2 -5502.16} C_VEL
LIN {X 0,Y 510.989,Z 333.296,A -85,B 0,C 180,E1 -5502.813,E2 -5502.813} C_VEL
LIN {X 0,Y 511.246,Z 321.315,A -85,B 0,C 180,E1 -5503.363,E2 -5503.363} C_VEL
LIN {X 0,Y 511.559,Z 307.477,A -85,B 0,C 180,E1 -5503.81,E2 -5503.81} C_VEL
LIN {X 0,Y 511.736,Z 294.745,A -85,B 0,C 180,E1 -5504.058,E2 -5504.058} C_VEL
LIN {X 0,Y 512.136,Z 205.897,A -85,B 0,C 180,E1 -5505.336,E2 -5505.336} C_VEL
LIN {X 0,Y 510.213,Z 193.274,A -85,B 0,C 180,E1 -5505.586,E2 -5505.586} C_VEL
LIN {X 0,Y 510.679,Z 174.096,A -85,B 0,C 180,E1 -5508.661,E2 -5508.661} C_VEL
LIN {X 0,Y 511.131,Z 156.099,A -85,B 0,C 180,E1 -5511.58,E2 -5511.58} C_VEL
LIN {X 0,Y 511.279,Z 147.899,A -85,B 0,C 180,E1 -5512.93,E2 -5512.93} C_VEL
LIN {X 0,Y 509.816,Z 139.981,A -85,B 0,C 180,E1 -5514.32,E2 -5514.32} C_VEL
LIN {X 0,Y 509.813,Z 139.983,A -85,B 0,C 180,E1 -5517.059,E2 -5517.059} C_VEL
LIN {X 0,Y 509.782,Z 139.988,A -85,B 0,C 180,E1 -5519.755,E2 -5519.755} C_VEL
LIN {X 0,Y 509.824,Z 139.98,A -85,B 0,C 180,E1 -5522.765,E2 -5522.765} C_VEL
LIN {X 0,Y 509.791,Z 139.983,A -85,B 0,C 180,E1 -5525.572,E2 -5525.572} C_VEL
LIN {X 0,Y 509.81,Z 139.979,A -85,B 0,C 180,E1 -5528.341,E2 -5528.341} C_VEL
LIN {X 0,Y 509.798,Z 139.983,A -85,B 0,C 180,E1 -5531.43,E2 -5531.43} C_VEL
LIN {X 0,Y 509.836,Z 139.98,A -85,B 0,C 180,E1 -5534.669,E2 -5534.669} C_VEL
LIN {X 0,Y 509.783,Z 139.98,A -85,B 0,C 180,E1 -5537.505,E2 -5537.505} C_VEL
LIN {X 0,Y 509.822,Z 139.98,A -85,B 0,C 180,E1 -5540.645,E2 -5540.645} C_VEL
LIN {X 0,Y 509.766,Z 139.98,A -85,B 0,C 180,E1 -5543.642,E2 -5543.642} C_VEL
LIN {X 0,Y 509.832,Z 139.979,A -85,B 0,C 180,E1 -5546.537,E2 -5546.537} C_VEL
LIN {X 0,Y 509.795,Z 139.977,A -85,B 0,C 180,E1 -5549.331,E2 -5549.331} C_VEL
LIN {X 0,Y 509.815,Z 139.978,A -85,B 0,C 180,E1 -5552.05,E2 -5552.05} C_VEL
LIN {X 0,Y 509.793,Z 139.985,A -85,B 0,C 180,E1 -5554.699,E2 -5554.699} C_VEL
LIN {X 0,Y 509.817,Z 139.972,A -85,B 0,C 180,E1 -5557.458,E2 -5557.458} C_VEL
LIN {X 0,Y 509.817,Z 139.978,A -85,B 0,C 180,E1 -5560.679,E2 -5560.679} C_VEL
LIN {X 0,Y 509.787,Z 139.98,A -85,B 0,C 180,E1 -5563.171,E2 -5563.171} C_VEL
LIN {X 0,Y 509.835,Z 139.973,A -85,B 0,C 180,E1 -5565.633,E2 -5565.633} C_VEL
LIN {X 0,Y 509.881,Z 139.973,A -85,B 0,C 180,E1 -5568.13,E2 -5568.13} C_VEL
LIN {X 0,Y 509.864,Z 139.969,A -85,B 0,C 180,E1 -5571.279,E2 -5571.279} C_VEL
LIN {X 0,Y 509.907,Z 139.968,A -85,B 0,C 180,E1 -5573.669,E2 -5573.669} C_VEL
LIN {X 0,Y 509.875,Z 139.969,A -85,B 0,C 180,E1 -5576.839,E2 -5576.839} C_VEL
LIN {X 0,Y 509.913,Z 139.967,A -85,B 0,C 180,E1 -5578.42,E2 -5578.42} C_VEL
LIN {X 0,Y 510.025,Z 139.957,A -85,B 0,C 180,E1 -5580,E2 -5580} C_VEL
LIN {X 0,Y 510.033,Z 139.951,A -85,B 0,C 180,E1 -5582.369,E2 -5582.369} C_VEL
LIN {X 0,Y 509.927,Z 139.967,A -85,B 0,C 180,E1 -5585.536,E2 -5585.536} C_VEL
LIN {X 0,Y 509.865,Z 139.978,A -85,B 0,C 180,E1 -5587.923,E2 -5587.923} C_VEL
LIN {X 0,Y 509.853,Z 139.975,A -85,B 0,C 180,E1 -5591.126,E2 -5591.126} C_VEL
LIN {X 0,Y 509.831,Z 139.984,A -85,B 0,C 180,E1 -5593.553,E2 -5593.553} C_VEL
LIN {X 0,Y 509.79,Z 139.985,A -85,B 0,C 180,E1 -5596.005,E2 -5596.005} C_VEL
LIN {X 0,Y 509.823,Z 139.977,A -85,B 0,C 180,E1 -5598.485,E2 -5598.485} C_VEL
LIN {X 0,Y 509.823,Z 139.981,A -85,B 0,C 180,E1 -5601.002,E2 -5601.002} C_VEL
LIN {X 0,Y 509.847,Z 140.109,A -85,B 0,C 180,E1 -5603.428,E2 -5603.428} C_VEL
LIN {X 0,Y 510.594,Z 145.126,A -85,B 0,C 180,E1 -5604.389,E2 -5604.389} C_VEL
LIN {X 0,Y 510.393,Z 160.754,A -85,B 0,C 180,E1 -5607.248,E2 -5607.248} C_VEL
LIN {X 0,Y 510.323,Z 167.43,A -85,B 0,C 180,E1 -5608.473,E2 -5608.473} C_VEL
LIN {X 0,Y 512.244,Z 178.077,A -85,B 0,C 180,E1 -5608.698,E2 -5608.698} C_VEL
LIN {X 0,Y 511.688,Z 274.684,A -85,B 0,C 180,E1 -5610.107,E2 -5610.107} C_VEL
LIN {X 0,Y 511.478,Z 288.021,A -85,B 0,C 180,E1 -5610.463,E2 -5610.463} C_VEL
LIN {X 0,Y 511.262,Z 300.832,A -85,B 0,C 180,E1 -5610.972,E2 -5610.972} C_VEL
LIN {X 0,Y 510.925,Z 312.919,A -85,B 0,C 180,E1 -5611.629,E2 -5611.629} C_VEL
LIN {X 0,Y 510.576,Z 324.832,A -85,B 0,C 180,E1 -5612.468,E2 -5612.468} C_VEL
LIN {X 0,Y 510.278,Z 334.037,A -85,B 0,C 180,E1 -5613.274,E2 -5613.274} C_VEL
LIN {X 0,Y 510.014,Z 343.03,A -85,B 0,C 180,E1 -5614.23,E2 -5614.23} C_VEL
LIN {X 0,Y 509.762,Z 351.809,A -85,B 0,C 180,E1 -5615.383,E2 -5615.383} C_VEL
LIN {X 0,Y 509.621,Z 356.065,A -85,B 0,C 180,E1 -5616.042,E2 -5616.042} C_VEL
LIN {X 0,Y 508.924,Z 359.349,A -85,B 0,C 180,E1 -5616.589,E2 -5616.589} C_VEL
LIN {X 0,Y 505.952,Z 364.267,A -85,B 0,C 180,E1 -5617.504,E2 -5617.504} C_VEL
LIN {X 0,Y 502.937,Z 368.439,A -85,B 0,C 180,E1 -5618.472,E2 -5618.472} C_VEL
LIN {X 0,Y 502.185,Z 370.558,A -85,B 0,C 180,E1 -5619.097,E2 -5619.097} C_VEL
LIN {X 0,Y 502.141,Z 373.364,A -85,B 0,C 180,E1 -5620.077,E2 -5620.077} C_VEL
LIN {X 0,Y 502.066,Z 375.656,A -85,B 0,C 180,E1 -5621.14,E2 -5621.14} C_VEL
LIN {X 0,Y 501.999,Z 377.255,A -85,B 0,C 180,E1 -5622.221,E2 -5622.221} C_VEL
LIN {X 0,Y 501.992,Z 378.115,A -85,B 0,C 180,E1 -5623.315,E2 -5623.315} C_VEL
LIN {X 0,Y 502.032,Z 378.206,A -85,B 0,C 180,E1 -5624.443,E2 -5624.443} C_VEL
LIN {X 0,Y 502.034,Z 377.523,A -85,B 0,C 180,E1 -5625.578,E2 -5625.578} C_VEL
LIN {X 0,Y 502.031,Z 376.046,A -85,B 0,C 180,E1 -5626.715,E2 -5626.715} C_VEL
LIN {X 0,Y 502.097,Z 373.644,A -85,B 0,C 180,E1 -5627.889,E2 -5627.889} C_VEL
LIN {X 0,Y 502.204,Z 370.218,A -85,B 0,C 180,E1 -5629.085,E2 -5629.085} C_VEL
LIN {X 0,Y 502.289,Z 365.59,A -85,B 0,C 180,E1 -5630.313,E2 -5630.313} C_VEL
LIN {X 0,Y 502.499,Z 359.603,A -85,B 0,C 180,E1 -5631.556,E2 -5631.556} C_VEL
LIN {X 0,Y 502.695,Z 351.862,A -85,B 0,C 180,E1 -5632.834,E2 -5632.834} C_VEL
LIN {X 0,Y 502.952,Z 343.568,A -85,B 0,C 180,E1 -5633.941,E2 -5633.941} C_VEL
LIN {X 0,Y 503.34,Z 334.192,A -85,B 0,C 180,E1 -5634.956,E2 -5634.956} C_VEL
LIN {X 0,Y 503.646,Z 323.944,A -85,B 0,C 180,E1 -5635.856,E2 -5635.856} C_VEL
LIN {X 0,Y 503.981,Z 312.45,A -85,B 0,C 180,E1 -5636.665,E2 -5636.665} C_VEL
LIN {X 0,Y 504.329,Z 300.451,A -85,B 0,C 180,E1 -5637.317,E2 -5637.317} C_VEL
LIN {X 0,Y 504.578,Z 286.916,A -85,B 0,C 180,E1 -5637.852,E2 -5637.852} C_VEL
LIN {X 0,Y 504.779,Z 274.261,A -85,B 0,C 180,E1 -5638.185,E2 -5638.185} C_VEL
LIN {X 0,Y 505.326,Z 178.628,A -85,B 0,C 180,E1 -5639.595,E2 -5639.595} C_VEL
LIN {X 0,Y 503.295,Z 167.518,A -85,B 0,C 180,E1 -5639.84,E2 -5639.84} C_VEL
LIN {X 0,Y 503.712,Z 151.438,A -85,B 0,C 180,E1 -5642.954,E2 -5642.954} C_VEL
LIN {X 0,Y 503.753,Z 146.458,A -85,B 0,C 180,E1 -5643.931,E2 -5643.931} C_VEL
LIN {X 0,Y 502.775,Z 140.86,A -85,B 0,C 180,E1 -5645.096,E2 -5645.096} C_VEL
LIN {X 0,Y 502.768,Z 140.856,A -85,B 0,C 180,E1 -5647.826,E2 -5647.826} C_VEL
LIN {X 0,Y 502.798,Z 140.857,A -85,B 0,C 180,E1 -5650.4,E2 -5650.4} C_VEL
LIN {X 0,Y 502.752,Z 140.858,A -85,B 0,C 180,E1 -5652.929,E2 -5652.929} C_VEL
LIN {X 0,Y 502.821,Z 140.846,A -85,B 0,C 180,E1 -5655.429,E2 -5655.429} C_VEL
LIN {X 0,Y 502.833,Z 140.849,A -85,B 0,C 180,E1 -5658.716,E2 -5658.716} C_VEL
LIN {X 0,Y 502.842,Z 140.848,A -85,B 0,C 180,E1 -5661.966,E2 -5661.966} C_VEL
LIN {X 0,Y 502.888,Z 140.844,A -85,B 0,C 180,E1 -5664.386,E2 -5664.386} C_VEL
LIN {X 0,Y 503.005,Z 140.825,A -85,B 0,C 180,E1 -5667.598,E2 -5667.598} C_VEL
LIN {X 0,Y 502.999,Z 140.832,A -85,B 0,C 180,E1 -5670,E2 -5670} C_VEL
LIN {X 0,Y 503.005,Z 140.827,A -85,B 0,C 180,E1 -5672.402,E2 -5672.402} C_VEL
LIN {X 0,Y 502.888,Z 140.842,A -85,B 0,C 180,E1 -5675.614,E2 -5675.614} C_VEL
LIN {X 0,Y 502.842,Z 140.851,A -85,B 0,C 180,E1 -5678.034,E2 -5678.034} C_VEL
LIN {X 0,Y 502.833,Z 140.847,A -85,B 0,C 180,E1 -5681.284,E2 -5681.284} C_VEL
LIN {X 0,Y 502.82,Z 140.847,A -85,B 0,C 180,E1 -5684.571,E2 -5684.571} C_VEL
LIN {X 0,Y 502.779,Z 140.857,A -85,B 0,C 180,E1 -5687.91,E2 -5687.91} C_VEL
LIN {X 0,Y 502.798,Z 140.849,A -85,B 0,C 180,E1 -5690.528,E2 -5690.528} C_VEL
LIN {X 0,Y 502.777,Z 140.854,A -85,B 0,C 180,E1 -5693.041,E2 -5693.041} C_VEL
LIN {X 0,Y 502.772,Z 140.859,A -85,B 0,C 180,E1 -5695.679,E2 -5695.679} C_VEL
LIN {X 0,Y 502.754,Z 140.855,A -85,B 0,C 180,E1 -5698.378,E2 -5698.378} C_VEL
LIN {X 0,Y 502.78,Z 140.859,A -85,B 0,C 180,E1 -5701.497,E2 -5701.497} C_VEL
LIN {X 0,Y 502.78,Z 140.852,A -85,B 0,C 180,E1 -5704.441,E2 -5704.441} C_VEL
LIN {X 0,Y 502.756,Z 140.862,A -85,B 0,C 180,E1 -5707.175,E2 -5707.175} C_VEL
LIN {X 0,Y 502.764,Z 140.854,A -85,B 0,C 180,E1 -5710.017,E2 -5710.017} C_VEL
LIN {X 0,Y 502.74,Z 140.864,A -85,B 0,C 180,E1 -5713.234,E2 -5713.234} C_VEL
LIN {X 0,Y 502.772,Z 140.854,A -85,B 0,C 180,E1 -5715.66,E2 -5715.66} C_VEL
LIN {X 0,Y 502.758,Z 140.863,A -85,B 0,C 180,E1 -5719.012,E2 -5719.012} C_VEL
LIN {X 0,Y 502.754,Z 140.855,A -85,B 0,C 180,E1 -5722.043,E2 -5722.043} C_VEL
LIN {X 0,Y 502.776,Z 140.858,A -85,B 0,C 180,E1 -5725.033,E2 -5725.033} C_VEL
LIN {X 0,Y 502.771,Z 140.853,A -85,B 0,C 180,E1 -5727.915,E2 -5727.915} C_VEL
LIN {X 0,Y 502.782,Z 140.86,A -85,B 0,C 180,E1 -5730.71,E2 -5730.71} C_VEL
LIN {X 0,Y 502.766,Z 140.854,A -85,B 0,C 180,E1 -5733.46,E2 -5733.46} C_VEL
LIN {X 0,Y 502.753,Z 140.857,A -85,B 0,C 180,E1 -5736.085,E2 -5736.085} C_VEL
LIN {X 0,Y 502.762,Z 140.861,A -85,B 0,C 180,E1 -5738.688,E2 -5738.688} C_VEL
LIN {X 0,Y 502.798,Z 140.85,A -85,B 0,C 180,E1 -5741.247,E2 -5741.247} C_VEL
LIN {X 0,Y 502.828,Z 140.851,A -85,B 0,C 180,E1 -5744.665,E2 -5744.665} C_VEL
LIN {X 0,Y 502.863,Z 140.846,A -85,B 0,C 180,E1 -5748.044,E2 -5748.044} C_VEL
LIN {X 0,Y 502.829,Z 140.846,A -85,B 0,C 180,E1 -5751.156,E2 -5751.156} C_VEL
LIN {X 0,Y 502.86,Z 140.843,A -85,B 0,C 180,E1 -5753.581,E2 -5753.581} C_VEL
LIN {X 0,Y 502.823,Z 140.847,A -85,B 0,C 180,E1 -5756.795,E2 -5756.795} C_VEL
LIN {X 0,Y 502.886,Z 140.843,A -85,B 0,C 180,E1 -5758.399,E2 -5758.399} C_VEL
LIN {X 0,Y 502.996,Z 140.833,A -85,B 0,C 180,E1 -5760,E2 -5760} C_VEL
LIN {X 0,Y 503.002,Z 140.827,A -85,B 0,C 180,E1 -5762.403,E2 -5762.403} C_VEL
LIN {X 0,Y 502.885,Z 140.843,A -85,B 0,C 180,E1 -5765.614,E2 -5765.614} C_VEL
LIN {X 0,Y 502.84,Z 140.851,A -85,B 0,C 180,E1 -5768.035,E2 -5768.035} C_VEL
LIN {X 0,Y 502.831,Z 140.847,A -85,B 0,C 180,E1 -5771.285,E2 -5771.285} C_VEL
LIN {X 0,Y 502.818,Z 140.847,A -85,B 0,C 180,E1 -5774.572,E2 -5774.572} C_VEL
LIN {X 0,Y 502.778,Z 140.857,A -85,B 0,C 180,E1 -5777.91,E2 -5777.91} C_VEL
LIN {X 0,Y 502.797,Z 140.849,A -85,B 0,C 180,E1 -5780.528,E2 -5780.528} C_VEL
LIN {X 0,Y 502.776,Z 140.854,A -85,B 0,C 180,E1 -5783.042,E2 -5783.042} C_VEL
LIN {X 0,Y 502.771,Z 140.859,A -85,B 0,C 180,E1 -5785.68,E2 -5785.68} C_VEL
LIN {X 0,Y 502.755,Z 140.855,A -85,B 0,C 180,E1 -5788.378,E2 -5788.378} C_VEL
LIN {X 0,Y 502.766,Z 140.86,A -85,B 0,C 180,E1 -5791.495,E2 -5791.495} C_VEL
LIN {X 0,Y 502.781,Z 140.852,A -85,B 0,C 180,E1 -5794.441,E2 -5794.441} C_VEL
LIN {X 0,Y 502.733,Z 140.866,A -85,B 0,C 180,E1 -5797.172,E2 -5797.172} C_VEL
LIN {X 0,Y 502.765,Z 140.854,A -85,B 0,C 180,E1 -5800.018,E2 -5800.018} C_VEL
LIN {X 0,Y 502.737,Z 140.864,A -85,B 0,C 180,E1 -5803.236,E2 -5803.236} C_VEL
LIN {X 0,Y 502.765,Z 140.855,A -85,B 0,C 180,E1 -5805.659,E2 -5805.659} C_VEL
LIN {X 0,Y 502.761,Z 140.862,A -85,B 0,C 180,E1 -5809.013,E2 -5809.013} C_VEL
LIN {X 0,Y 502.757,Z 140.855,A -85,B 0,C 180,E1 -5812.043,E2 -5812.043} C_VEL
LIN {X 0,Y 502.78,Z 140.857,A -85,B 0,C 180,E1 -5815.033,E2 -5815.033} C_VEL
LIN {X 0,Y 502.757,Z 140.855,A -85,B 0,C 180,E1 -5817.914,E2 -5817.914} C_VEL
LIN {X 0,Y 502.752,Z 140.863,A -85,B 0,C 180,E1 -5820.708,E2 -5820.708} C_VEL
LIN {X 0,Y 502.77,Z 140.853,A -85,B 0,C 180,E1 -5823.461,E2 -5823.461} C_VEL
LIN {X 0,Y 502.791,Z 140.982,A -85,B 0,C 180,E1 -5825.348,E2 -5825.348} C_VEL
LIN {X 0,Y 504.451,Z 150.374,A -85,B 0,C 180,E1 -5827.04,E2 -5827.04} C_VEL
LIN {X 0,Y 504.092,Z 163.98,A -85,B 0,C 180,E1 -5829.332,E2 -5829.332} C_VEL
LIN {X 0,Y 503.605,Z 179.585,A -85,B 0,C 180,E1 -5831.924,E2 -5831.924} C_VEL
LIN {X 0,Y 503.256,Z 193.443,A -85,B 0,C 180,E1 -5834.201,E2 -5834.201} C_VEL
LIN {X 0,Y 505.32,Z 208.164,A -85,B 0,C 180,E1 -5834.487,E2 -5834.487} C_VEL
LIN {X 0,Y 504.766,Z 301.941,A -85,B 0,C 180,E1 -5835.872,E2 -5835.872} C_VEL
LIN {X 0,Y 504.483,Z 315.793,A -85,B 0,C 180,E1 -5836.249,E2 -5836.249} C_VEL
LIN {X 0,Y 504.142,Z 328.233,A -85,B 0,C 180,E1 -5836.753,E2 -5836.753} C_VEL
LIN {X 0,Y 503.762,Z 340.912,A -85,B 0,C 180,E1 -5837.459,E2 -5837.459} C_VEL
LIN {X 0,Y 503.471,Z 352.879,A -85,B 0,C 180,E1 -5838.322,E2 -5838.322} C_VEL
LIN {X 0,Y 503.169,Z 361.908,A -85,B 0,C 180,E1 -5839.131,E2 -5839.131} C_VEL
LIN {X 0,Y 502.813,Z 371.169,A -85,B 0,C 180,E1 -5840.141,E2 -5840.141} C_VEL
LIN {X 0,Y 502.554,Z 380.174,A -85,B 0,C 180,E1 -5841.354,E2 -5841.354} C_VEL
LIN {X 0,Y 502.344,Z 387.425,A -85,B 0,C 180,E1 -5842.564,E2 -5842.564} C_VEL
LIN {X 0,Y 502.236,Z 392.317,A -85,B 0,C 180,E1 -5843.572,E2 -5843.572} C_VEL
LIN {X 0,Y 502.172,Z 397.07,A -85,B 0,C 180,E1 -5844.781,E2 -5844.781} C_VEL
LIN {X 0,Y 502.137,Z 400.7,A -85,B 0,C 180,E1 -5845.987,E2 -5845.987} C_VEL
LIN {X 0,Y 502.12,Z 402.573,A -85,B 0,C 180,E1 -5846.79,E2 -5846.79} C_VEL
LIN {X 0,Y 502.092,Z 403.976,A -85,B 0,C 180,E1 -5847.593,E2 -5847.593} C_VEL
LIN {X 0,Y 501.993,Z 405.58,A -85,B 0,C 180,E1 -5849.198,E2 -5849.198} C_VEL
LIN {X 0,Y 501.984,Z 405.795,A -85,B 0,C 180,E1 -5850,E2 -5850} C_VEL
LIN {X 0,Y 502.036,Z 404.959,A -85,B 0,C 180,E1 -5851.604,E2 -5851.604} C_VEL
LIN {X 0,Y 502.092,Z 403.954,A -85,B 0,C 180,E1 -5852.407,E2 -5852.407} C_VEL
LIN {X 0,Y 502.12,Z 402.543,A -85,B 0,C 180,E1 -5853.209,E2 -5853.209} C_VEL
LIN {X 0,Y 502.1,Z 399.579,A -85,B 0,C 180,E1 -5854.415,E2 -5854.415} C_VEL
LIN {X 0,Y 502.199,Z 395.57,A -85,B 0,C 180,E1 -5855.622,E2 -5855.622} C_VEL
LIN {X 0,Y 502.327,Z 389.5,A -85,B 0,C 180,E1 -5857.011,E2 -5857.011} C_VEL
LIN {X 0,Y 502.47,Z 382.657,A -85,B 0,C 180,E1 -5858.242,E2 -5858.242} C_VEL
LIN {X 0,Y 502.706,Z 374.295,A -85,B 0,C 180,E1 -5859.454,E2 -5859.454} C_VEL
LIN {X 0,Y 502.958,Z 365.697,A -85,B 0,C 180,E1 -5860.466,E2 -5860.466} C_VEL
LIN {X 0,Y 503.347,Z 355.086,A -85,B 0,C 180,E1 -5861.476,E2 -5861.476} C_VEL
LIN {X 0,Y 503.658,Z 343.939,A -85,B 0,C 180,E1 -5862.331,E2 -5862.331} C_VEL
LIN {X 0,Y 504.041,Z 332.994,A -85,B 0,C 180,E1 -5862.993,E2 -5862.993} C_VEL
LIN {X 0,Y 504.309,Z 320.979,A -85,B 0,C 180,E1 -5863.55,E2 -5863.55} C_VEL
LIN {X 0,Y 504.645,Z 308.01,A -85,B 0,C 180,E1 -5863.977,E2 -5863.977} C_VEL
LIN {X 0,Y 504.847,Z 294.224,A -85,B 0,C 180,E1 -5864.254,E2 -5864.254} C_VEL
LIN {X 0,Y 505.32,Z 206.973,A -85,B 0,C 180,E1 -5865.53,E2 -5865.53} C_VEL
LIN {X 0,Y 503.204,Z 193.012,A -85,B 0,C 180,E1 -5865.817,E2 -5865.817} C_VEL
LIN {X 0,Y 503.731,Z 173.876,A -85,B 0,C 180,E1 -5868.928,E2 -5868.928} C_VEL
LIN {X 0,Y 504.18,Z 157.185,A -85,B 0,C 180,E1 -5871.678,E2 -5871.678} C_VEL
LIN {X 0,Y 504.259,Z 148.723,A -85,B 0,C 180,E1 -5873.094,E2 -5873.094} C_VEL
LIN {X 0,Y 502.769,Z 140.86,A -85,B 0,C 180,E1 -5874.505,E2 -5874.505} C_VEL
LIN {X 0,Y 502.767,Z 140.865,A -85,B 0,C 180,E1 -5877.47,E2 -5877.47} C_VEL
LIN {X 0,Y 502.741,Z 140.863,A -85,B 0,C 180,E1 -5880.215,E2 -5880.215} C_VEL
LIN {X 0,Y 502.797,Z 140.858,A -85,B 0,C 180,E1 -5883.033,E2 -5883.033} C_VEL
LIN {X 0,Y 502.742,Z 140.859,A -85,B 0,C 180,E1 -5885.953,E2 -5885.953} C_VEL
LIN {X 0,Y 502.777,Z 140.861,A -85,B 0,C 180,E1 -5888.977,E2 -5888.977} C_VEL
LIN {X 0,Y 502.741,Z 140.86,A -85,B 0,C 180,E1 -5892.191,E2 -5892.191} C_VEL
LIN {X 0,Y 502.774,Z 140.856,A -85,B 0,C 180,E1 -5895.47,E2 -5895.47} C_VEL
LIN {X 0,Y 502.756,Z 140.863,A -85,B 0,C 180,E1 -5898.927,E2 -5898.927} C_VEL
LIN {X 0,Y 502.755,Z 140.856,A -85,B 0,C 180,E1 -5902.042,E2 -5902.042} C_VEL
LIN {X 0,Y 502.777,Z 140.857,A -85,B 0,C 180,E1 -5905.032,E2 -5905.032} C_VEL
LIN {X 0,Y 502.766,Z 140.854,A -85,B 0,C 180,E1 -5907.914,E2 -5907.914} C_VEL
LIN {X 0,Y 502.745,Z 140.862,A -85,B 0,C 180,E1 -5910.707,E2 -5910.707} C_VEL
LIN {X 0,Y 502.767,Z 140.851,A -85,B 0,C 180,E1 -5913.459,E2 -5913.459} C_VEL
LIN {X 0,Y 502.753,Z 140.859,A -85,B 0,C 180,E1 -5916.084,E2 -5916.084} C_VEL
LIN {X 0,Y 502.751,Z 140.861,A -85,B 0,C 180,E1 -5918.687,E2 -5918.687} C_VEL
LIN {X 0,Y 502.785,Z 140.852,A -85,B 0,C 180,E1 -5921.896,E2 -5921.896} C_VEL
LIN {X 0,Y 502.828,Z 140.848,A -85,B 0,C 180,E1 -5924.664,E2 -5924.664} C_VEL
LIN {X 0,Y 502.862,Z 140.848,A -85,B 0,C 180,E1 -5928.043,E2 -5928.043} C_VEL
LIN {X 0,Y 502.828,Z 140.846,A -85,B 0,C 180,E1 -5931.156,E2 -5931.156} C_VEL
LIN {X 0,Y 502.858,Z 140.845,A -85,B 0,C 180,E1 -5933.58,E2 -5933.58} C_VEL
LIN {X 0,Y 502.821,Z 140.848,A -85,B 0,C 180,E1 -5936.795,E2 -5936.795} C_VEL
LIN {X 0,Y 502.883,Z 140.843,A -85,B 0,C 180,E1 -5938.398,E2 -5938.398} C_VEL
LIN {X 0,Y 502.994,Z 140.832,A -85,B 0,C 180,E1 -5940,E2 -5940} C_VEL
LIN {X 0,Y 503,Z 140.827,A -85,B 0,C 180,E1 -5942.402,E2 -5942.402} C_VEL
LIN {X 0,Y 502.883,Z 140.846,A -85,B 0,C 180,E1 -5945.614,E2 -5945.614} C_VEL
LIN {X 0,Y 502.837,Z 140.852,A -85,B 0,C 180,E1 -5948.034,E2 -5948.034} C_VEL
LIN {X 0,Y 502.828,Z 140.852,A -85,B 0,C 180,E1 -5951.284,E2 -5951.284} C_VEL
LIN {X 0,Y 502.816,Z 140.852,A -85,B 0,C 180,E1 -5954.571,E2 -5954.571} C_VEL
LIN {X 0,Y 502.785,Z 140.855,A -85,B 0,C 180,E1 -5958.103,E2 -5958.103} C_VEL
LIN {X 0,Y 502.821,Z 140.851,A -85,B 0,C 180,E1 -5960.536,E2 -5960.536} C_VEL
LIN {X 0,Y 502.819,Z 140.901,A -85,B 0,C 180,E1 -5963.257,E2 -5963.257} C_VEL
LIN {X 0,Y 503.652,Z 146.348,A -85,B 0,C 180,E1 -5964.308,E2 -5964.308} C_VEL
LIN {X 0,Y 503.411,Z 162.085,A -85,B 0,C 180,E1 -5967.224,E2 -5967.224} C_VEL
LIN {X 0,Y 503.336,Z 167.617,A -85,B 0,C 180,E1 -5968.248,E2 -5968.248} C_VEL
LIN {X 0,Y 505.465,Z 179.757,A -85,B 0,C 180,E1 -5968.507,E2 -5968.507} C_VEL
LIN {X 0,Y 504.781,Z 275.736,A -85,B 0,C 180,E1 -5969.937,E2 -5969.937} C_VEL
LIN {X 0,Y 504.543,Z 289.291,A -85,B 0,C 180,E1 -5970.314,E2 -5970.314} C_VEL
LIN {X 0,Y 504.321,Z 301.801,A -85,B 0,C 180,E1 -5970.832,E2 -5970.832} C_VEL
LIN {X 0,Y 503.996,Z 313.394,A -85,B 0,C 180,E1 -5971.478,E2 -5971.478} C_VEL
LIN {X 0,Y 503.641,Z 324.382,A -85,B 0,C 180,E1 -5972.259,E2 -5972.259} C_VEL
LIN {X 0,Y 503.296,Z 333.841,A -85,B 0,C 180,E1 -5973.089,E2 -5973.089} C_VEL
LIN {X 0,Y 503.009,Z 343.224,A -85,B 0,C 180,E1 -5974.095,E2 -5974.095} C_VEL
LIN {X 0,Y 502.728,Z 351.409,A -85,B 0,C 180,E1 -5975.175,E2 -5975.175} C_VEL
LIN {X 0,Y 502.475,Z 359.342,A -85,B 0,C 180,E1 -5976.472,E2 -5976.472} C_VEL
LIN {X 0,Y 502.343,Z 365.579,A -85,B 0,C 180,E1 -5977.759,E2 -5977.759} C_VEL
LIN {X 0,Y 502.185,Z 370.558,A -85,B 0,C 180,E1 -5979.097,E2 -5979.097} C_VEL
LIN {X 0,Y 501.452,Z 372.493,A -85,B 0,C 180,E1 -5979.733,E2 -5979.733} C_VEL
LIN {X 0,Y 498.511,Z 375.124,A -85,B 0,C 180,E1 -5980.776,E2 -5980.776} C_VEL
LIN {X 0,Y 496.052,Z 376.712,A -85,B 0,C 180,E1 -5981.63,E2 -5981.63} C_VEL
LIN {X 0,Y 494.989,Z 377.553,A -85,B 0,C 180,E1 -5982.298,E2 -5982.298} C_VEL
LIN {X 0,Y 494.898,Z 377.754,A -85,B 0,C 180,E1 -5982.526,E2 -5982.526} C_VEL
LIN {X 0,Y 494.921,Z 378.474,A -85,B 0,C 180,E1 -5984.091,E2 -5984.091} C_VEL
LIN {X 0,Y 494.941,Z 378.031,A -85,B 0,C 180,E1 -5985.233,E2 -5985.233} C_VEL
LIN {X 0,Y 494.923,Z 376.764,A -85,B 0,C 180,E1 -5986.403,E2 -5986.403} C_VEL
LIN {X 0,Y 494.998,Z 374.627,A -85,B 0,C 180,E1 -5987.586,E2 -5987.586} C_VEL
LIN {X 0,Y 495.122,Z 370.133,A -85,B 0,C 180,E1 -5989.237,E2 -5989.237} C_VEL
LIN {X 0,Y 495.263,Z 365.013,A -85,B 0,C 180,E1 -5990.573,E2 -5990.573} C_VEL
LIN {X 0,Y 495.453,Z 358.473,A -85,B 0,C 180,E1 -5991.9,E2 -5991.9} C_VEL
LIN {X 0,Y 495.667,Z 351.632,A -85,B 0,C 180,E1 -5993.017,E2 -5993.017} C_VEL
LIN {X 0,Y 495.942,Z 344.025,A -85,B 0,C 180,E1 -5994.041,E2 -5994.041} C_VEL
LIN {X 0,Y 496.344,Z 334.55,A -85,B 0,C 180,E1 -5995.088,E2 -5995.088} C_VEL
LIN {X 0,Y 496.687,Z 324.092,A -85,B 0,C 180,E1 -5996.02,E2 -5996.02} C_VEL
LIN {X 0,Y 497.002,Z 313.613,A -85,B 0,C 180,E1 -5996.774,E2 -5996.774} C_VEL
LIN {X 0,Y 497.398,Z 301.318,A -85,B 0,C 180,E1 -5997.466,E2 -5997.466} C_VEL
LIN {X 0,Y 497.678,Z 288.331,A -85,B 0,C 180,E1 -5997.999,E2 -5997.999} C_VEL
LIN {X 0,Y 497.89,Z 274.808,A -85,B 0,C 180,E1 -5998.37,E2 -5998.37} C_VEL
LIN {X 0,Y 498.504,Z 179.58,A -85,B 0,C 180,E1 -5999.8,E2 -5999.8} C_VEL
LIN {X 0,Y 496.299,Z 167.715,A -85,B 0,C 180,E1 -6000.061,E2 -6000.061} C_VEL
LIN {X 0,Y 496.798,Z 151.123,A -85,B 0,C 180,E1 -6003.311,E2 -6003.311} C_VEL
LIN {X 0,Y 496.65,Z 146.652,A -85,B 0,C 180,E1 -6004.207,E2 -6004.207} C_VEL
LIN {X 0,Y 495.746,Z 141.735,A -85,B 0,C 180,E1 -6005.269,E2 -6005.269} C_VEL
LIN {X 0,Y 495.727,Z 141.738,A -85,B 0,C 180,E1 -6008.371,E2 -6008.371} C_VEL
LIN {X 0,Y 495.759,Z 141.729,A -85,B 0,C 180,E1 -6010.971,E2 -6010.971} C_VEL
LIN {X 0,Y 495.798,Z 141.728,A -85,B 0,C 180,E1 -6014.558,E2 -6014.558} C_VEL
LIN {X 0,Y 495.818,Z 141.722,A -85,B 0,C 180,E1 -6017.97,E2 -6017.97} C_VEL
LIN {X 0,Y 495.789,Z 141.723,A -85,B 0,C 180,E1 -6021.03,E2 -6021.03} C_VEL
LIN {X 0,Y 495.814,Z 141.72,A -85,B 0,C 180,E1 -6023.489,E2 -6023.489} C_VEL
LIN {X 0,Y 495.7,Z 141.739,A -85,B 0,C 180,E1 -6025.935,E2 -6025.935} C_VEL
LIN {X 0,Y 495.971,Z 141.701,A -85,B 0,C 180,E1 -6027.564,E2 -6027.564} C_VEL
LIN {X 0,Y 495.968,Z 141.708,A -85,B 0,C 180,E1 -6030,E2 -6030} C_VEL
LIN {X 0,Y 495.971,Z 141.703,A -85,B 0,C 180,E1 -6032.437,E2 -6032.437} C_VEL
LIN {X 0,Y 495.846,Z 141.72,A -85,B 0,C 180,E1 -6035.694,E2 -6035.694} C_VEL
LIN {X 0,Y 495.806,Z 141.725,A -85,B 0,C 180,E1 -6038.149,E2 -6038.149} C_VEL
LIN {X 0,Y 495.818,Z 141.722,A -85,B 0,C 180,E1 -6041.446,E2 -6041.446} C_VEL
LIN {X 0,Y 495.771,Z 141.725,A -85,B 0,C 180,E1 -6044.783,E2 -6044.783} C_VEL
LIN {X 0,Y 495.743,Z 141.73,A -85,B 0,C 180,E1 -6048.226,E2 -6048.226} C_VEL
LIN {X 0,Y 495.742,Z 141.729,A -85,B 0,C 180,E1 -6050.758,E2 -6050.758} C_VEL
LIN {X 0,Y 495.729,Z 141.736,A -85,B 0,C 180,E1 -6053.388,E2 -6053.388} C_VEL
LIN {X 0,Y 495.712,Z 141.734,A -85,B 0,C 180,E1 -6056.072,E2 -6056.072} C_VEL
LIN {X 0,Y 495.69,Z 141.736,A -85,B 0,C 180,E1 -6058.82,E2 -6058.82} C_VEL
LIN {X 0,Y 495.744,Z 141.732,A -85,B 0,C 180,E1 -6061.724,E2 -6061.724} C_VEL
LIN {X 0,Y 495.752,Z 141.728,A -85,B 0,C 180,E1 -6064.692,E2 -6064.692} C_VEL
LIN {X 0,Y 495.707,Z 141.737,A -85,B 0,C 180,E1 -6067.563,E2 -6067.563} C_VEL
LIN {X 0,Y 495.736,Z 141.729,A -85,B 0,C 180,E1 -6070.045,E2 -6070.045} C_VEL
LIN {X 0,Y 495.689,Z 141.74,A -85,B 0,C 180,E1 -6072.886,E2 -6072.886} C_VEL
LIN {X 0,Y 495.716,Z 141.732,A -85,B 0,C 180,E1 -6075.998,E2 -6075.998} C_VEL
LIN {X 0,Y 495.72,Z 141.735,A -85,B 0,C 180,E1 -6079.296,E2 -6079.296} C_VEL
LIN {X 0,Y 495.717,Z 141.734,A -85,B 0,C 180,E1 -6081.406,E2 -6081.406} C_VEL
LIN {X 0,Y 495.722,Z 141.734,A -85,B 0,C 180,E1 -6084.461,E2 -6084.461} C_VEL
LIN {X 0,Y 495.743,Z 141.73,A -85,B 0,C 180,E1 -6087.404,E2 -6087.404} C_VEL
LIN {X 0,Y 495.732,Z 141.732,A -85,B 0,C 180,E1 -6090.252,E2 -6090.252} C_VEL
LIN {X 0,Y 495.731,Z 141.731,A -85,B 0,C 180,E1 -6093.271,E2 -6093.271} C_VEL
LIN {X 0,Y 495.701,Z 141.733,A -85,B 0,C 180,E1 -6095.723,E2 -6095.723} C_VEL
LIN {X 0,Y 495.725,Z 141.737,A -85,B 0,C 180,E1 -6098.371,E2 -6098.371} C_VEL
LIN {X 0,Y 495.756,Z 141.729,A -85,B 0,C 180,E1 -6100.971,E2 -6100.971} C_VEL
LIN {X 0,Y 495.796,Z 141.728,A -85,B 0,C 180,E1 -6104.558,E2 -6104.558} C_VEL
LIN {X 0,Y 495.815,Z 141.723,A -85,B 0,C 180,E1 -6107.97,E2 -6107.97} C_VEL
LIN {X 0,Y 495.77,Z 141.725,A -85,B 0,C 180,E1 -6111.029,E2 -6111.029} C_VEL
LIN {X 0,Y 495.811,Z 141.72,A -85,B 0,C 180,E1 -6113.489,E2 -6113.489} C_VEL
LIN {X 0,Y 495.697,Z 141.739,A -85,B 0,C 180,E1 -6115.935,E2 -6115.935} C_VEL
LIN {X 0,Y 495.968,Z 141.702,A -85,B 0,C 180,E1 -6117.564,E2 -6117.564} C_VEL
LIN {X 0,Y 495.965,Z 141.708,A -85,B 0,C 180,E1 -6120,E2 -6120} C_VEL
LIN {X 0,Y 495.969,Z 141.703,A -85,B 0,C 180,E1 -6122.437,E2 -6122.437} C_VEL
LIN {X 0,Y 495.844,Z 141.721,A -85,B 0,C 180,E1 -6125.694,E2 -6125.694} C_VEL
LIN {X 0,Y 495.804,Z 141.725,A -85,B 0,C 180,E1 -6128.149,E2 -6128.149} C_VEL
LIN {X 0,Y 495.816,Z 141.723,A -85,B 0,C 180,E1 -6131.446,E2 -6131.446} C_VEL
LIN {X 0,Y 495.769,Z 141.725,A -85,B 0,C 180,E1 -6134.784,E2 -6134.784} C_VEL
LIN {X 0,Y 495.742,Z 141.73,A -85,B 0,C 180,E1 -6138.226,E2 -6138.226} C_VEL
LIN {X 0,Y 495.741,Z 141.729,A -85,B 0,C 180,E1 -6140.758,E2 -6140.758} C_VEL
LIN {X 0,Y 495.729,Z 141.737,A -85,B 0,C 180,E1 -6143.389,E2 -6143.389} C_VEL
LIN {X 0,Y 495.711,Z 141.734,A -85,B 0,C 180,E1 -6146.073,E2 -6146.073} C_VEL
LIN {X 0,Y 495.691,Z 141.736,A -85,B 0,C 180,E1 -6148.82,E2 -6148.82} C_VEL
LIN {X 0,Y 495.733,Z 141.733,A -85,B 0,C 180,E1 -6151.722,E2 -6151.722} C_VEL
LIN {X 0,Y 495.751,Z 141.729,A -85,B 0,C 180,E1 -6154.692,E2 -6154.692} C_VEL
LIN {X 0,Y 495.697,Z 141.738,A -85,B 0,C 180,E1 -6157.565,E2 -6157.565} C_VEL
LIN {X 0,Y 495.738,Z 141.729,A -85,B 0,C 180,E1 -6160.045,E2 -6160.045} C_VEL
LIN {X 0,Y 495.688,Z 141.741,A -85,B 0,C 180,E1 -6162.888,E2 -6162.888} C_VEL
LIN {X 0,Y 495.711,Z 141.732,A -85,B 0,C 180,E1 -6165.997,E2 -6165.997} C_VEL
LIN {X 0,Y 495.724,Z 141.734,A -85,B 0,C 180,E1 -6169.296,E2 -6169.296} C_VEL
LIN {X 0,Y 495.72,Z 141.733,A -85,B 0,C 180,E1 -6171.406,E2 -6171.406} C_VEL
LIN {X 0,Y 495.726,Z 141.734,A -85,B 0,C 180,E1 -6174.461,E2 -6174.461} C_VEL
LIN {X 0,Y 495.74,Z 141.73,A -85,B 0,C 180,E1 -6177.404,E2 -6177.404} C_VEL
LIN {X 0,Y 495.695,Z 141.737,A -85,B 0,C 180,E1 -6180.249,E2 -6180.249} C_VEL
LIN {X 0,Y 495.721,Z 141.732,A -85,B 0,C 180,E1 -6183.275,E2 -6183.275} C_VEL
LIN {X 0,Y 495.724,Z 141.74,A -85,B 0,C 180,E1 -6185.141,E2 -6185.141} C_VEL
LIN {X 0,Y 497.48,Z 150.984,A -85,B 0,C 180,E1 -6186.838,E2 -6186.838} C_VEL
LIN {X 0,Y 497.186,Z 163.695,A -85,B 0,C 180,E1 -6189.016,E2 -6189.016} C_VEL
LIN {X 0,Y 496.607,Z 180.585,A -85,B 0,C 180,E1 -6191.86,E2 -6191.86} C_VEL
LIN {X 0,Y 496.253,Z 193.201,A -85,B 0,C 180,E1 -6193.964,E2 -6193.964} C_VEL
LIN {X 0,Y 498.483,Z 207.848,A -85,B 0,C 180,E1 -6194.268,E2 -6194.268} C_VEL
LIN {X 0,Y 497.89,Z 301.467,A -85,B 0,C 180,E1 -6195.673,E2 -6195.673} C_VEL
LIN {X 0,Y 497.61,Z 314.646,A -85,B 0,C 180,E1 -6196.029,E2 -6196.029} C_VEL
LIN {X 0,Y 497.279,Z 326.783,A -85,B 0,C 180,E1 -6196.515,E2 -6196.515} C_VEL
LIN {X 0,Y 496.91,Z 338.415,A -85,B 0,C 180,E1 -6197.14,E2 -6197.14} C_VEL
LIN {X 0,Y 496.517,Z 350.012,A -85,B 0,C 180,E1 -6197.949,E2 -6197.949} C_VEL
LIN {X 0,Y 496.211,Z 360.582,A -85,B 0,C 180,E1 -6198.874,E2 -6198.874} C_VEL
LIN {X 0,Y 495.826,Z 369.216,A -85,B 0,C 180,E1 -6199.795,E2 -6199.795} C_VEL
LIN {X 0,Y 495.586,Z 377.179,A -85,B 0,C 180,E1 -6200.82,E2 -6200.82} C_VEL
LIN {X 0,Y 495.33,Z 384.96,A -85,B 0,C 180,E1 -6202.048,E2 -6202.048} C_VEL
LIN {X 0,Y 495.18,Z 390.274,A -85,B 0,C 180,E1 -6203.071,E2 -6203.071} C_VEL
LIN {X 0,Y 495.117,Z 395.43,A -85,B 0,C 180,E1 -6204.298,E2 -6204.298} C_VEL
LIN {X 0,Y 495.006,Z 399.425,A -85,B 0,C 180,E1 -6205.521,E2 -6205.521} C_VEL
LIN {X 0,Y 495.042,Z 402.376,A -85,B 0,C 180,E1 -6206.745,E2 -6206.745} C_VEL
LIN {X 0,Y 494.998,Z 403.781,A -85,B 0,C 180,E1 -6207.559,E2 -6207.559} C_VEL
LIN {X 0,Y 494.963,Z 404.779,A -85,B 0,C 180,E1 -6208.373,E2 -6208.373} C_VEL
LIN {X 0,Y 494.902,Z 405.601,A -85,B 0,C 180,E1 -6210,E2 -6210} C_VEL
LIN {X 0,Y 494.963,Z 404.762,A -85,B 0,C 180,E1 -6211.627,E2 -6211.627} C_VEL
LIN {X 0,Y 494.998,Z 403.755,A -85,B 0,C 180,E1 -6212.441,E2 -6212.441} C_VEL
LIN {X 0,Y 495.042,Z 402.342,A -85,B 0,C 180,E1 -6213.255,E2 -6213.255} C_VEL
LIN {X 0,Y 495.006,Z 399.374,A -85,B 0,C 180,E1 -6214.478,E2 -6214.478} C_VEL
LIN {X 0,Y 495.115,Z 395.36,A -85,B 0,C 180,E1 -6215.702,E2 -6215.702} C_VEL
LIN {X 0,Y 495.253,Z 389.18,A -85,B 0,C 180,E1 -6217.133,E2 -6217.133} C_VEL
LIN {X 0,Y 495.418,Z 382.432,A -85,B 0,C 180,E1 -6218.361,E2 -6218.361} C_VEL
LIN {X 0,Y 495.683,Z 374.06,A -85,B 0,C 180,E1 -6219.59,E2 -6219.59} C_VEL
LIN {X 0,Y 495.96,Z 365.449,A -85,B 0,C 180,E1 -6220.615,E2 -6220.615} C_VEL
LIN {X 0,Y 496.353,Z 354.823,A -85,B 0,C 180,E1 -6221.64,E2 -6221.64} C_VEL
LIN {X 0,Y 496.683,Z 343.947,A -85,B 0,C 180,E1 -6222.487,E2 -6222.487} C_VEL
LIN {X 0,Y 497.097,Z 332.707,A -85,B 0,C 180,E1 -6223.178,E2 -6223.178} C_VEL
LIN {X 0,Y 497.408,Z 320.678,A -85,B 0,C 180,E1 -6223.742,E2 -6223.742} C_VEL
LIN {X 0,Y 497.738,Z 307.688,A -85,B 0,C 180,E1 -6224.175,E2 -6224.175} C_VEL
LIN {X 0,Y 497.974,Z 293.84,A -85,B 0,C 180,E1 -6224.455,E2 -6224.455} C_VEL
LIN {X 0,Y 498.34,Z 206.612,A -85,B 0,C 180,E1 -6225.758,E2 -6225.758} C_VEL
LIN {X 0,Y 496.22,Z 192.815,A -85,B 0,C 180,E1 -6226.046,E2 -6226.046} C_VEL
LIN {X 0,Y 496.772,Z 173.694,A -85,B 0,C 180,E1 -6229.203,E2 -6229.203} C_VEL
LIN {X 0,Y 497.241,Z 158.273,A -85,B 0,C 180,E1 -6231.778,E2 -6231.778} C_VEL
LIN {X 0,Y 497.363,Z 150.316,A -85,B 0,C 180,E1 -6233.124,E2 -6233.124} C_VEL
LIN {X 0,Y 495.729,Z 141.738,A -85,B 0,C 180,E1 -6234.696,E2 -6234.696} C_VEL
LIN {X 0,Y 495.708,Z 141.739,A -85,B 0,C 180,E1 -6237.895,E2 -6237.895} C_VEL
LIN {X 0,Y 495.707,Z 141.741,A -85,B 0,C 180,E1 -6240.69,E2 -6240.69} C_VEL
LIN {X 0,Y 495.736,Z 141.735,A -85,B 0,C 180,E1 -6243.565,E2 -6243.565} C_VEL
LIN {X 0,Y 495.685,Z 141.739,A -85,B 0,C 180,E1 -6246.547,E2 -6246.547} C_VEL
LIN {X 0,Y 495.737,Z 141.734,A -85,B 0,C 180,E1 -6249.639,E2 -6249.639} C_VEL
LIN {X 0,Y 495.691,Z 141.743,A -85,B 0,C 180,E1 -6252.886,E2 -6252.886} C_VEL
LIN {X 0,Y 495.709,Z 141.734,A -85,B 0,C 180,E1 -6255.996,E2 -6255.996} C_VEL
LIN {X 0,Y 495.72,Z 141.734,A -85,B 0,C 180,E1 -6259.295,E2 -6259.295} C_VEL
LIN {X 0,Y 495.717,Z 141.734,A -85,B 0,C 180,E1 -6261.405,E2 -6261.405} C_VEL
LIN {X 0,Y 495.724,Z 141.734,A -85,B 0,C 180,E1 -6264.46,E2 -6264.46} C_VEL
LIN {X 0,Y 495.742,Z 141.729,A -85,B 0,C 180,E1 -6267.403,E2 -6267.403} C_VEL
LIN {X 0,Y 495.689,Z 141.737,A -85,B 0,C 180,E1 -6270.248,E2 -6270.248} C_VEL
LIN {X 0,Y 495.732,Z 141.728,A -85,B 0,C 180,E1 -6273.27,E2 -6273.27} C_VEL
LIN {X 0,Y 495.702,Z 141.735,A -85,B 0,C 180,E1 -6275.722,E2 -6275.722} C_VEL
LIN {X 0,Y 495.718,Z 141.736,A -85,B 0,C 180,E1 -6278.37,E2 -6278.37} C_VEL
LIN {X 0,Y 495.742,Z 141.728,A -85,B 0,C 180,E1 -6280.97,E2 -6280.97} C_VEL
LIN {X 0,Y 495.795,Z 141.725,A -85,B 0,C 180,E1 -6284.557,E2 -6284.557} C_VEL
LIN {X 0,Y 495.814,Z 141.725,A -85,B 0,C 180,E1 -6287.969,E2 -6287.969} C_VEL
LIN {X 0,Y 495.785,Z 141.723,A -85,B 0,C 180,E1 -6291.029,E2 -6291.029} C_VEL
LIN {X 0,Y 495.809,Z 141.722,A -85,B 0,C 180,E1 -6293.488,E2 -6293.488} C_VEL
LIN {X 0,Y 495.695,Z 141.74,A -85,B 0,C 180,E1 -6295.935,E2 -6295.935} C_VEL
LIN {X 0,Y 495.967,Z 141.704,A -85,B 0,C 180,E1 -6297.563,E2 -6297.563} C_VEL
LIN {X 0,Y 495.963,Z 141.708,A -85,B 0,C 180,E1 -6300,E2 -6300} C_VEL
LIN {X 0,Y 495.967,Z 141.703,A -85,B 0,C 180,E1 -6302.436,E2 -6302.436} C_VEL
LIN {X 0,Y 495.842,Z 141.723,A -85,B 0,C 180,E1 -6305.694,E2 -6305.694} C_VEL
LIN {X 0,Y 495.801,Z 141.727,A -85,B 0,C 180,E1 -6308.149,E2 -6308.149} C_VEL
LIN {X 0,Y 495.813,Z 141.728,A -85,B 0,C 180,E1 -6311.446,E2 -6311.446} C_VEL
LIN {X 0,Y 495.767,Z 141.73,A -85,B 0,C 180,E1 -6314.783,E2 -6314.783} C_VEL
LIN {X 0,Y 495.763,Z 141.729,A -85,B 0,C 180,E1 -6318.235,E2 -6318.235} C_VEL
LIN {X 0,Y 495.764,Z 141.731,A -85,B 0,C 180,E1 -6320.756,E2 -6320.756} C_VEL
LIN {X 0,Y 495.771,Z 141.853,A -85,B 0,C 180,E1 -6323.115,E2 -6323.115} C_VEL
LIN {X 0,Y 496.701,Z 147.568,A -85,B 0,C 180,E1 -6324.225,E2 -6324.225} C_VEL
LIN {X 0,Y 496.446,Z 162.023,A -85,B 0,C 180,E1 -6326.937,E2 -6326.937} C_VEL
LIN {X 0,Y 496.359,Z 167.827,A -85,B 0,C 180,E1 -6328.021,E2 -6328.021} C_VEL
LIN {X 0,Y 498.625,Z 180.638,A -85,B 0,C 180,E1 -6328.296,E2 -6328.296} C_VEL
LIN {X 0,Y 497.91,Z 275.764,A -85,B 0,C 180,E1 -6329.736,E2 -6329.736} C_VEL
LIN {X 0,Y 497.654,Z 289.355,A -85,B 0,C 180,E1 -6330.118,E2 -6330.118} C_VEL
LIN {X 0,Y 497.434,Z 301.655,A -85,B 0,C 180,E1 -6330.631,E2 -6330.631} C_VEL
LIN {X 0,Y 497.065,Z 313.624,A -85,B 0,C 180,E1 -6331.306,E2 -6331.306} C_VEL
LIN {X 0,Y 496.687,Z 324.493,A -85,B 0,C 180,E1 -6332.088,E2 -6332.088} C_VEL
LIN {X 0,Y 496.288,Z 335.084,A -85,B 0,C 180,E1 -6333.038,E2 -6333.038} C_VEL
LIN {X 0,Y 495.931,Z 345.051,A -85,B 0,C 180,E1 -6334.162,E2 -6334.162} C_VEL
LIN {X 0,Y 495.629,Z 353.375,A -85,B 0,C 180,E1 -6335.319,E2 -6335.319} C_VEL
LIN {X 0,Y 495.389,Z 360.648,A -85,B 0,C 180,E1 -6336.573,E2 -6336.573} C_VEL
LIN {X 0,Y 495.239,Z 366.546,A -85,B 0,C 180,E1 -6337.862,E2 -6337.862} C_VEL
LIN {X 0,Y 495.108,Z 371.197,A -85,B 0,C 180,E1 -6339.173,E2 -6339.173} C_VEL
LIN {X 0,Y 495.046,Z 373.378,A -85,B 0,C 180,E1 -6339.95,E2 -6339.95} C_VEL
LIN {X 0,Y 494.988,Z 376.019,A -85,B 0,C 180,E1 -6341.193,E2 -6341.193} C_VEL
LIN {X 0,Y 494.898,Z 377.754,A -85,B 0,C 180,E1 -6342.526,E2 -6342.526} C_VEL
LIN {X 0,Y 494.215,Z 378.28,A -85,B 0,C 180,E1 -6343.204,E2 -6343.204} C_VEL
LIN {X 0,Y 491.348,Z 378.57,A -85,B 0,C 180,E1 -6344.31,E2 -6344.31} C_VEL
LIN {X 0,Y 488.946,Z 378.295,A -85,B 0,C 180,E1 -6345.199,E2 -6345.199} C_VEL
LIN {X 0,Y 487.928,Z 377.686,A -85,B 0,C 180,E1 -6345.882,E2 -6345.882} C_VEL
LIN {X 0,Y 487.853,Z 377.396,A -85,B 0,C 180,E1 -6346.112,E2 -6346.112} C_VEL
LIN {X 0,Y 487.901,Z 375.347,A -85,B 0,C 180,E1 -6347.39,E2 -6347.39} C_VEL
LIN {X 0,Y 487.987,Z 372.699,A -85,B 0,C 180,E1 -6348.511,E2 -6348.511} C_VEL
LIN {X 0,Y 488.08,Z 368.824,A -85,B 0,C 180,E1 -6349.743,E2 -6349.743} C_VEL
LIN {X 0,Y 488.254,Z 363.673,A -85,B 0,C 180,E1 -6351.012,E2 -6351.012} C_VEL
LIN {X 0,Y 488.451,Z 356.967,A -85,B 0,C 180,E1 -6352.312,E2 -6352.312} C_VEL
LIN {X 0,Y 488.795,Z 348.419,A -85,B 0,C 180,E1 -6353.627,E2 -6353.627} C_VEL
LIN {X 0,Y 489.129,Z 340.082,A -85,B 0,C 180,E1 -6354.668,E2 -6354.668} C_VEL
LIN {X 0,Y 489.508,Z 329.918,A -85,B 0,C 180,E1 -6355.701,E2 -6355.701} C_VEL
LIN {X 0,Y 489.94,Z 318.268,A -85,B 0,C 180,E1 -6356.642,E2 -6356.642} C_VEL
LIN {X 0,Y 490.29,Z 306.645,A -85,B 0,C 180,E1 -6357.382,E2 -6357.382} C_VEL
LIN {X 0,Y 490.697,Z 293.564,A -85,B 0,C 180,E1 -6358,E2 -6358} C_VEL
LIN {X 0,Y 490.912,Z 280.449,A -85,B 0,C 180,E1 -6358.438,E2 -6358.438} C_VEL
LIN {X 0,Y 491.106,Z 267.766,A -85,B 0,C 180,E1 -6358.692,E2 -6358.692} C_VEL
LIN {X 0,Y 491.656,Z 180.358,A -85,B 0,C 180,E1 -6360.01,E2 -6360.01} C_VEL
LIN {X 0,Y 489.316,Z 167.845,A -85,B 0,C 180,E1 -6360.297,E2 -6360.297} C_VEL
LIN {X 0,Y 489.883,Z 151.2,A -85,B 0,C 180,E1 -6363.594,E2 -6363.594} C_VEL
LIN {X 0,Y 489.478,Z 146.862,A -85,B 0,C 180,E1 -6364.486,E2 -6364.486} C_VEL
LIN {X 0,Y 488.682,Z 142.614,A -85,B 0,C 180,E1 -6365.408,E2 -6365.408} C_VEL
LIN {X 0,Y 488.682,Z 142.613,A -85,B 0,C 180,E1 -6368.043,E2 -6368.043} C_VEL
LIN {X 0,Y 488.722,Z 142.611,A -85,B 0,C 180,E1 -6370.686,E2 -6370.686} C_VEL
LIN {X 0,Y 488.671,Z 142.609,A -85,B 0,C 180,E1 -6373.284,E2 -6373.284} C_VEL
LIN {X 0,Y 488.716,Z 142.605,A -85,B 0,C 180,E1 -6375.85,E2 -6375.85} C_VEL
LIN {X 0,Y 488.78,Z 142.604,A -85,B 0,C 180,E1 -6378.387,E2 -6378.387} C_VEL
LIN {X 0,Y 488.753,Z 142.601,A -85,B 0,C 180,E1 -6381.733,E2 -6381.733} C_VEL
LIN {X 0,Y 488.806,Z 142.601,A -85,B 0,C 180,E1 -6384.224,E2 -6384.224} C_VEL
LIN {X 0,Y 488.937,Z 142.577,A -85,B 0,C 180,E1 -6387.529,E2 -6387.529} C_VEL
LIN {X 0,Y 488.937,Z 142.583,A -85,B 0,C 180,E1 -6390,E2 -6390} C_VEL
LIN {X 0,Y 488.937,Z 142.579,A -85,B 0,C 180,E1 -6392.472,E2 -6392.472} C_VEL
LIN {X 0,Y 488.806,Z 142.598,A -85,B 0,C 180,E1 -6395.776,E2 -6395.776} C_VEL
LIN {X 0,Y 488.753,Z 142.603,A -85,B 0,C 180,E1 -6398.267,E2 -6398.267} C_VEL
LIN {X 0,Y 488.78,Z 142.601,A -85,B 0,C 180,E1 -6401.613,E2 -6401.613} C_VEL
LIN {X 0,Y 488.742,Z 142.601,A -85,B 0,C 180,E1 -6405.001,E2 -6405.001} C_VEL
LIN {X 0,Y 488.702,Z 142.606,A -85,B 0,C 180,E1 -6408.444,E2 -6408.444} C_VEL
LIN {X 0,Y 488.685,Z 142.609,A -85,B 0,C 180,E1 -6411.072,E2 -6411.072} C_VEL
LIN {X 0,Y 488.66,Z 142.616,A -85,B 0,C 180,E1 -6413.747,E2 -6413.747} C_VEL
LIN {X 0,Y 488.677,Z 142.609,A -85,B 0,C 180,E1 -6416.476,E2 -6416.476} C_VEL
LIN {X 0,Y 488.661,Z 142.617,A -85,B 0,C 180,E1 -6419.274,E2 -6419.274} C_VEL
LIN {X 0,Y 488.69,Z 142.607,A -85,B 0,C 180,E1 -6422.148,E2 -6422.148} C_VEL
LIN {X 0,Y 488.705,Z 142.611,A -85,B 0,C 180,E1 -6425.116,E2 -6425.116} C_VEL
LIN {X 0,Y 488.656,Z 142.611,A -85,B 0,C 180,E1 -6428.202,E2 -6428.202} C_VEL
LIN {X 0,Y 488.688,Z 142.607,A -85,B 0,C 180,E1 -6430.341,E2 -6430.341} C_VEL
LIN {X 0,Y 488.667,Z 142.612,A -85,B 0,C 180,E1 -6433.656,E2 -6433.656} C_VEL
LIN {X 0,Y 488.667,Z 142.611,A -85,B 0,C 180,E1 -6436.344,E2 -6436.344} C_VEL
LIN {X 0,Y 488.697,Z 142.607,A -85,B 0,C 180,E1 -6439.674,E2 -6439.674} C_VEL
LIN {X 0,Y 488.644,Z 142.62,A -85,B 0,C 180,E1 -6442.838,E2 -6442.838} C_VEL
LIN {X 0,Y 488.709,Z 142.604,A -85,B 0,C 180,E1 -6445.886,E2 -6445.886} C_VEL
LIN {X 0,Y 488.675,Z 142.617,A -85,B 0,C 180,E1 -6448.82,E2 -6448.82} C_VEL
LIN {X 0,Y 488.684,Z 142.608,A -85,B 0,C 180,E1 -6451.668,E2 -6451.668} C_VEL
LIN {X 0,Y 488.682,Z 142.613,A -85,B 0,C 180,E1 -6454.441,E2 -6454.441} C_VEL
LIN {X 0,Y 488.7,Z 142.607,A -85,B 0,C 180,E1 -6457.152,E2 -6457.152} C_VEL
LIN {X 0,Y 488.704,Z 142.606,A -85,B 0,C 180,E1 -6459.81,E2 -6459.81} C_VEL
LIN {X 0,Y 488.666,Z 142.618,A -85,B 0,C 180,E1 -6462.421,E2 -6462.421} C_VEL
LIN {X 0,Y 488.74,Z 142.602,A -85,B 0,C 180,E1 -6464.999,E2 -6464.999} C_VEL
LIN {X 0,Y 488.777,Z 142.604,A -85,B 0,C 180,E1 -6468.387,E2 -6468.387} C_VEL
LIN {X 0,Y 488.747,Z 142.602,A -85,B 0,C 180,E1 -6471.733,E2 -6471.733} C_VEL
LIN {X 0,Y 488.803,Z 142.601,A -85,B 0,C 180,E1 -6474.224,E2 -6474.224} C_VEL
LIN {X 0,Y 488.934,Z 142.578,A -85,B 0,C 180,E1 -6477.529,E2 -6477.529} C_VEL
LIN {X 0,Y 488.934,Z 142.584,A -85,B 0,C 180,E1 -6480,E2 -6480} C_VEL
LIN {X 0,Y 488.934,Z 142.579,A -85,B 0,C 180,E1 -6482.472,E2 -6482.472} C_VEL
LIN {X 0,Y 488.803,Z 142.599,A -85,B 0,C 180,E1 -6485.777,E2 -6485.777} C_VEL
LIN {X 0,Y 488.75,Z 142.603,A -85,B 0,C 180,E1 -6488.268,E2 -6488.268} C_VEL
LIN {X 0,Y 488.778,Z 142.602,A -85,B 0,C 180,E1 -6491.613,E2 -6491.613} C_VEL
LIN {X 0,Y 488.74,Z 142.601,A -85,B 0,C 180,E1 -6495.001,E2 -6495.001} C_VEL
LIN {X 0,Y 488.701,Z 142.606,A -85,B 0,C 180,E1 -6498.445,E2 -6498.445} C_VEL
LIN {X 0,Y 488.685,Z 142.61,A -85,B 0,C 180,E1 -6501.072,E2 -6501.072} C_VEL
LIN {X 0,Y 488.66,Z 142.616,A -85,B 0,C 180,E1 -6503.748,E2 -6503.748} C_VEL
LIN {X 0,Y 488.677,Z 142.608,A -85,B 0,C 180,E1 -6506.477,E2 -6506.477} C_VEL
LIN {X 0,Y 488.654,Z 142.618,A -85,B 0,C 180,E1 -6509.275,E2 -6509.275} C_VEL
LIN {X 0,Y 488.686,Z 142.608,A -85,B 0,C 180,E1 -6512.149,E2 -6512.149} C_VEL
LIN {X 0,Y 488.702,Z 142.612,A -85,B 0,C 180,E1 -6515.117,E2 -6515.117} C_VEL
LIN {X 0,Y 488.652,Z 142.612,A -85,B 0,C 180,E1 -6518.203,E2 -6518.203} C_VEL
LIN {X 0,Y 488.691,Z 142.607,A -85,B 0,C 180,E1 -6520.342,E2 -6520.342} C_VEL
LIN {X 0,Y 488.663,Z 142.612,A -85,B 0,C 180,E1 -6523.658,E2 -6523.658} C_VEL
LIN {X 0,Y 488.663,Z 142.611,A -85,B 0,C 180,E1 -6526.344,E2 -6526.344} C_VEL
LIN {X 0,Y 488.703,Z 142.606,A -85,B 0,C 180,E1 -6529.674,E2 -6529.674} C_VEL
LIN {X 0,Y 488.647,Z 142.62,A -85,B 0,C 180,E1 -6532.839,E2 -6532.839} C_VEL
LIN {X 0,Y 488.714,Z 142.604,A -85,B 0,C 180,E1 -6535.886,E2 -6535.886} C_VEL
LIN {X 0,Y 488.658,Z 142.619,A -85,B 0,C 180,E1 -6538.818,E2 -6538.818} C_VEL
LIN {X 0,Y 488.684,Z 142.609,A -85,B 0,C 180,E1 -6541.668,E2 -6541.668} C_VEL
LIN {X 0,Y 488.692,Z 142.656,A -85,B 0,C 180,E1 -6544.961,E2 -6544.961} C_VEL
LIN {X 0,Y 490.572,Z 153.088,A -85,B 0,C 180,E1 -6546.899,E2 -6546.899} C_VEL
LIN {X 0,Y 490.063,Z 167.728,A -85,B 0,C 180,E1 -6549.43,E2 -6549.43} C_VEL
LIN {X 0,Y 489.608,Z 181.645,A -85,B 0,C 180,E1 -6551.808,E2 -6551.808} C_VEL
LIN {X 0,Y 489.266,Z 193.257,A -85,B 0,C 180,E1 -6553.748,E2 -6553.748} C_VEL
LIN {X 0,Y 491.649,Z 208.743,A -85,B 0,C 180,E1 -6554.065,E2 -6554.065} C_VEL
LIN {X 0,Y 490.998,Z 302.057,A -85,B 0,C 180,E1 -6555.494,E2 -6555.494} C_VEL
LIN {X 0,Y 490.682,Z 315.737,A -85,B 0,C 180,E1 -6555.881,E2 -6555.881} C_VEL
LIN {X 0,Y 490.336,Z 327.545,A -85,B 0,C 180,E1 -6556.373,E2 -6556.373} C_VEL
LIN {X 0,Y 489.887,Z 340.013,A -85,B 0,C 180,E1 -6557.078,E2 -6557.078} C_VEL
LIN {X 0,Y 489.512,Z 351.029,A -85,B 0,C 180,E1 -6557.879,E2 -6557.879} C_VEL
LIN {X 0,Y 489.184,Z 361.395,A -85,B 0,C 180,E1 -6558.817,E2 -6558.817} C_VEL
LIN {X 0,Y 488.736,Z 370.69,A -85,B 0,C 180,E1 -6559.854,E2 -6559.854} C_VEL
LIN {X 0,Y 488.421,Z 379.718,A -85,B 0,C 180,E1 -6561.102,E2 -6561.102} C_VEL
LIN {X 0,Y 488.206,Z 386.988,A -85,B 0,C 180,E1 -6562.348,E2 -6562.348} C_VEL
LIN {X 0,Y 488.048,Z 392.507,A -85,B 0,C 180,E1 -6563.524,E2 -6563.524} C_VEL
LIN {X 0,Y 488.014,Z 396.66,A -85,B 0,C 180,E1 -6564.629,E2 -6564.629} C_VEL
LIN {X 0,Y 487.926,Z 400.298,A -85,B 0,C 180,E1 -6565.87,E2 -6565.87} C_VEL
LIN {X 0,Y 487.964,Z 402.178,A -85,B 0,C 180,E1 -6566.697,E2 -6566.697} C_VEL
LIN {X 0,Y 487.909,Z 403.584,A -85,B 0,C 180,E1 -6567.523,E2 -6567.523} C_VEL
LIN {X 0,Y 487.891,Z 404.584,A -85,B 0,C 180,E1 -6568.349,E2 -6568.349} C_VEL
LIN {X 0,Y 487.823,Z 405.407,A -85,B 0,C 180,E1 -6570,E2 -6570} C_VEL
LIN {X 0,Y 487.891,Z 404.567,A -85,B 0,C 180,E1 -6571.651,E2 -6571.651} C_VEL
LIN {X 0,Y 487.909,Z 403.558,A -85,B 0,C 180,E1 -6572.477,E2 -6572.477} C_VEL
LIN {X 0,Y 487.964,Z 402.143,A -85,B 0,C 180,E1 -6573.302,E2 -6573.302} C_VEL
LIN {X 0,Y 487.918,Z 399.17,A -85,B 0,C 180,E1 -6574.544,E2 -6574.544} C_VEL
LIN {X 0,Y 488.011,Z 395.151,A -85,B 0,C 180,E1 -6575.786,E2 -6575.786} C_VEL
LIN {X 0,Y 488.179,Z 388.964,A -85,B 0,C 180,E1 -6577.236,E2 -6577.236} C_VEL
LIN {X 0,Y 488.35,Z 382.211,A -85,B 0,C 180,E1 -6578.482,E2 -6578.482} C_VEL
LIN {X 0,Y 488.651,Z 373.835,A -85,B 0,C 180,E1 -6579.729,E2 -6579.729} C_VEL
LIN {X 0,Y 488.973,Z 365.219,A -85,B 0,C 180,E1 -6580.769,E2 -6580.769} C_VEL
LIN {X 0,Y 489.378,Z 354.59,A -85,B 0,C 180,E1 -6581.808,E2 -6581.808} C_VEL
LIN {X 0,Y 489.759,Z 342.905,A -85,B 0,C 180,E1 -6582.724,E2 -6582.724} C_VEL
LIN {X 0,Y 490.242,Z 330.459,A -85,B 0,C 180,E1 -6583.471,E2 -6583.471} C_VEL
LIN {X 0,Y 490.595,Z 317.81,A -85,B 0,C 180,E1 -6584.042,E2 -6584.042} C_VEL
LIN {X 0,Y 490.936,Z 305.487,A -85,B 0,C 180,E1 -6584.429,E2 -6584.429} C_VEL
LIN {X 0,Y 491.155,Z 290.036,A -85,B 0,C 180,E1 -6584.713,E2 -6584.713} C_VEL
LIN {X 0,Y 491.594,Z 207.77,A -85,B 0,C 180,E1 -6585.964,E2 -6585.964} C_VEL
LIN {X 0,Y 489.22,Z 192.593,A -85,B 0,C 180,E1 -6586.289,E2 -6586.289} C_VEL
LIN {X 0,Y 489.791,Z 173.512,A -85,B 0,C 180,E1 -6589.488,E2 -6589.488} C_VEL
LIN {X 0,Y 490.372,Z 156.805,A -85,B 0,C 180,E1 -6592.321,E2 -6592.321} C_VEL
LIN {X 0,Y 490.466,Z 152.338,A -85,B 0,C 180,E1 -6593.088,E2 -6593.088} C_VEL
LIN {X 0,Y 488.682,Z 142.615,A -85,B 0,C 180,E1 -6594.895,E2 -6594.895} C_VEL
LIN {X 0,Y 488.674,Z 142.62,A -85,B 0,C 180,E1 -6597.401,E2 -6597.401} C_VEL
LIN {X 0,Y 488.65,Z 142.619,A -85,B 0,C 180,E1 -6600.35,E2 -6600.35} C_VEL
LIN {X 0,Y 488.706,Z 142.611,A -85,B 0,C 180,E1 -6603.478,E2 -6603.478} C_VEL
LIN {X 0,Y 488.646,Z 142.615,A -85,B 0,C 180,E1 -6606.348,E2 -6606.348} C_VEL
LIN {X 0,Y 488.682,Z 142.617,A -85,B 0,C 180,E1 -6609.255,E2 -6609.255} C_VEL
LIN {X 0,Y 488.663,Z 142.615,A -85,B 0,C 180,E1 -6611.593,E2 -6611.593} C_VEL
LIN {X 0,Y 488.696,Z 142.614,A -85,B 0,C 180,E1 -6614.802,E2 -6614.802} C_VEL
LIN {X 0,Y 488.644,Z 142.614,A -85,B 0,C 180,E1 -6617.469,E2 -6617.469} C_VEL
LIN {X 0,Y 488.7,Z 142.606,A -85,B 0,C 180,E1 -6619.673,E2 -6619.673} C_VEL
LIN {X 0,Y 488.645,Z 142.618,A -85,B 0,C 180,E1 -6622.838,E2 -6622.838} C_VEL
LIN {X 0,Y 488.711,Z 142.605,A -85,B 0,C 180,E1 -6625.885,E2 -6625.885} C_VEL
LIN {X 0,Y 488.656,Z 142.616,A -85,B 0,C 180,E1 -6628.817,E2 -6628.817} C_VEL
LIN {X 0,Y 488.678,Z 142.609,A -85,B 0,C 180,E1 -6631.667,E2 -6631.667} C_VEL
LIN {X 0,Y 488.683,Z 142.612,A -85,B 0,C 180,E1 -6634.44,E2 -6634.44} C_VEL
LIN {X 0,Y 488.7,Z 142.603,A -85,B 0,C 180,E1 -6637.152,E2 -6637.152} C_VEL
LIN {X 0,Y 488.685,Z 142.61,A -85,B 0,C 180,E1 -6639.808,E2 -6639.808} C_VEL
LIN {X 0,Y 488.665,Z 142.618,A -85,B 0,C 180,E1 -6642.421,E2 -6642.421} C_VEL
LIN {X 0,Y 488.738,Z 142.6,A -85,B 0,C 180,E1 -6644.999,E2 -6644.999} C_VEL
LIN {X 0,Y 488.776,Z 142.601,A -85,B 0,C 180,E1 -6648.387,E2 -6648.387} C_VEL
LIN {X 0,Y 488.748,Z 142.603,A -85,B 0,C 180,E1 -6651.732,E2 -6651.732} C_VEL
LIN {X 0,Y 488.802,Z 142.598,A -85,B 0,C 180,E1 -6654.223,E2 -6654.223} C_VEL
LIN {X 0,Y 488.933,Z 142.58,A -85,B 0,C 180,E1 -6657.528,E2 -6657.528} C_VEL
LIN {X 0,Y 488.932,Z 142.584,A -85,B 0,C 180,E1 -6660,E2 -6660} C_VEL
LIN {X 0,Y 488.933,Z 142.579,A -85,B 0,C 180,E1 -6662.471,E2 -6662.471} C_VEL
LIN {X 0,Y 488.801,Z 142.6,A -85,B 0,C 180,E1 -6665.776,E2 -6665.776} C_VEL
LIN {X 0,Y 488.747,Z 142.605,A -85,B 0,C 180,E1 -6668.267,E2 -6668.267} C_VEL
LIN {X 0,Y 488.775,Z 142.606,A -85,B 0,C 180,E1 -6671.613,E2 -6671.613} C_VEL
LIN {X 0,Y 488.737,Z 142.607,A -85,B 0,C 180,E1 -6675.001,E2 -6675.001} C_VEL
LIN {X 0,Y 488.735,Z 142.604,A -85,B 0,C 180,E1 -6678.443,E2 -6678.443} C_VEL
LIN {X 0,Y 488.695,Z 142.614,A -85,B 0,C 180,E1 -6681.071,E2 -6681.071} C_VEL
LIN {X 0,Y 488.723,Z 142.648,A -85,B 0,C 180,E1 -6682.931,E2 -6682.931} C_VEL
LIN {X 0,Y 489.738,Z 148.746,A -85,B 0,C 180,E1 -6684.141,E2 -6684.141} C_VEL
LIN {X 0,Y 489.452,Z 164.412,A -85,B 0,C 180,E1 -6687.097,E2 -6687.097} C_VEL
LIN {X 0,Y 489.371,Z 167.941,A -85,B 0,C 180,E1 -6687.764,E2 -6687.764} C_VEL
LIN {X 0,Y 491.801,Z 181.631,A -85,B 0,C 180,E1 -6688.079,E2 -6688.079} C_VEL
LIN {X 0,Y 491.07,Z 275.636,A -85,B 0,C 180,E1 -6689.526,E2 -6689.526} C_VEL
LIN {X 0,Y 490.81,Z 289.055,A -85,B 0,C 180,E1 -6689.904,E2 -6689.904} C_VEL
LIN {X 0,Y 490.523,Z 301.879,A -85,B 0,C 180,E1 -6690.441,E2 -6690.441} C_VEL
LIN {X 0,Y 490.18,Z 313.05,A -85,B 0,C 180,E1 -6691.074,E2 -6691.074} C_VEL
LIN {X 0,Y 489.757,Z 323.571,A -85,B 0,C 180,E1 -6691.827,E2 -6691.827} C_VEL
LIN {X 0,Y 489.317,Z 334.799,A -85,B 0,C 180,E1 -6692.833,E2 -6692.833} C_VEL
LIN {X 0,Y 488.98,Z 344.634,A -85,B 0,C 180,E1 -6693.942,E2 -6693.942} C_VEL
LIN {X 0,Y 488.638,Z 353.095,A -85,B 0,C 180,E1 -6695.121,E2 -6695.121} C_VEL
LIN {X 0,Y 488.371,Z 360.005,A -85,B 0,C 180,E1 -6696.306,E2 -6696.306} C_VEL
LIN {X 0,Y 488.196,Z 366.263,A -85,B 0,C 180,E1 -6697.65,E2 -6697.65} C_VEL
LIN {X 0,Y 488.04,Z 370.961,A -85,B 0,C 180,E1 -6698.958,E2 -6698.958} C_VEL
LIN {X 0,Y 487.915,Z 374.77,A -85,B 0,C 180,E1 -6700.404,E2 -6700.404} C_VEL
LIN {X 0,Y 487.88,Z 376.787,A -85,B 0,C 180,E1 -6701.501,E2 -6701.501} C_VEL
LIN {X 0,Y 487.798,Z 378.165,A -85,B 0,C 180,E1 -6702.712,E2 -6702.712} C_VEL
LIN {X 0,Y 487.829,Z 378.655,A -85,B 0,C 180,E1 -6703.919,E2 -6703.919} C_VEL
LIN {X 0,Y 487.858,Z 378.312,A -85,B 0,C 180,E1 -6705.1,E2 -6705.1} C_VEL
LIN {X 0,Y 487.853,Z 377.396,A -85,B 0,C 180,E1 -6706.112,E2 -6706.112} C_VEL
LIN {X 0,Y 487.214,Z 376.448,A -85,B 0,C 180,E1 -6706.792,E2 -6706.792} C_VEL
LIN {X 0,Y 484.406,Z 374.416,A -85,B 0,C 180,E1 -6707.889,E2 -6707.889} C_VEL
LIN {X 0,Y 482.047,Z 372.325,A -85,B 0,C 180,E1 -6708.757,E2 -6708.757} C_VEL
LIN {X 0,Y 481.062,Z 370.388,A -85,B 0,C 180,E1 -6709.414,E2 -6709.414} C_VEL
LIN {X 0,Y 480.998,Z 369.641,A -85,B 0,C 180,E1 -6709.633,E2 -6709.633} C_VEL
LIN {X 0,Y 481.183,Z 363.913,A -85,B 0,C 180,E1 -6711.095,E2 -6711.095} C_VEL
LIN {X 0,Y 481.407,Z 357.026,A -85,B 0,C 180,E1 -6712.447,E2 -6712.447} C_VEL
LIN {X 0,Y 481.775,Z 348.408,A -85,B 0,C 180,E1 -6713.787,E2 -6713.787} C_VEL
LIN {X 0,Y 482.192,Z 339.504,A -85,B 0,C 180,E1 -6714.902,E2 -6714.902} C_VEL
LIN {X 0,Y 482.603,Z 328.864,A -85,B 0,C 180,E1 -6715.972,E2 -6715.972} C_VEL
LIN {X 0,Y 482.988,Z 318.592,A -85,B 0,C 180,E1 -6716.806,E2 -6716.806} C_VEL
LIN {X 0,Y 483.394,Z 306.721,A -85,B 0,C 180,E1 -6717.572,E2 -6717.572} C_VEL
LIN {X 0,Y 483.795,Z 294.455,A -85,B 0,C 180,E1 -6718.164,E2 -6718.164} C_VEL
LIN {X 0,Y 484.023,Z 281.506,A -85,B 0,C 180,E1 -6718.611,E2 -6718.611} C_VEL
LIN {X 0,Y 484.225,Z 268.299,A -85,B 0,C 180,E1 -6718.89,E2 -6718.89} C_VEL
LIN {X 0,Y 484.94,Z 181.911,A -85,B 0,C 180,E1 -6720.211,E2 -6720.211} C_VEL
LIN {X 0,Y 482.36,Z 168.017,A -85,B 0,C 180,E1 -6720.532,E2 -6720.532} C_VEL
LIN {X 0,Y 482.909,Z 151.302,A -85,B 0,C 180,E1 -6723.881,E2 -6723.881} C_VEL
LIN {X 0,Y 481.659,Z 143.489,A -85,B 0,C 180,E1 -6725.571,E2 -6725.571} C_VEL
LIN {X 0,Y 481.683,Z 143.484,A -85,B 0,C 180,E1 -6729.033,E2 -6729.033} C_VEL
LIN {X 0,Y 481.661,Z 143.486,A -85,B 0,C 180,E1 -6732.157,E2 -6732.157} C_VEL
LIN {X 0,Y 481.724,Z 143.478,A -85,B 0,C 180,E1 -6734.776,E2 -6734.776} C_VEL
LIN {X 0,Y 481.731,Z 143.48,A -85,B 0,C 180,E1 -6738.215,E2 -6738.215} C_VEL
LIN {X 0,Y 481.711,Z 143.477,A -85,B 0,C 180,E1 -6741.611,E2 -6741.611} C_VEL
LIN {X 0,Y 481.768,Z 143.476,A -85,B 0,C 180,E1 -6744.139,E2 -6744.139} C_VEL
LIN {X 0,Y 481.903,Z 143.453,A -85,B 0,C 180,E1 -6747.493,E2 -6747.493} C_VEL
LIN {X 0,Y 481.906,Z 143.459,A -85,B 0,C 180,E1 -6750,E2 -6750} C_VEL
LIN {X 0,Y 481.903,Z 143.455,A -85,B 0,C 180,E1 -6752.508,E2 -6752.508} C_VEL
LIN {X 0,Y 481.768,Z 143.476,A -85,B 0,C 180,E1 -6755.861,E2 -6755.861} C_VEL
LIN {X 0,Y 481.712,Z 143.478,A -85,B 0,C 180,E1 -6758.389,E2 -6758.389} C_VEL
LIN {X 0,Y 481.732,Z 143.482,A -85,B 0,C 180,E1 -6761.785,E2 -6761.785} C_VEL
LIN {X 0,Y 481.725,Z 143.477,A -85,B 0,C 180,E1 -6765.225,E2 -6765.225} C_VEL
LIN {X 0,Y 481.645,Z 143.484,A -85,B 0,C 180,E1 -6768.724,E2 -6768.724} C_VEL
LIN {X 0,Y 481.625,Z 143.492,A -85,B 0,C 180,E1 -6771.395,E2 -6771.395} C_VEL
LIN {X 0,Y 481.641,Z 143.487,A -85,B 0,C 180,E1 -6774.115,E2 -6774.115} C_VEL
LIN {X 0,Y 481.646,Z 143.488,A -85,B 0,C 180,E1 -6777.116,E2 -6777.116} C_VEL
LIN {X 0,Y 481.603,Z 143.494,A -85,B 0,C 180,E1 -6779.746,E2 -6779.746} C_VEL
LIN {X 0,Y 481.646,Z 143.485,A -85,B 0,C 180,E1 -6782.676,E2 -6782.676} C_VEL
LIN {X 0,Y 481.623,Z 143.49,A -85,B 0,C 180,E1 -6785.71,E2 -6785.71} C_VEL
LIN {X 0,Y 481.627,Z 143.49,A -85,B 0,C 180,E1 -6788.863,E2 -6788.863} C_VEL
LIN {X 0,Y 481.615,Z 143.489,A -85,B 0,C 180,E1 -6791.908,E2 -6791.908} C_VEL
LIN {X 0,Y 481.648,Z 143.485,A -85,B 0,C 180,E1 -6794.458,E2 -6794.458} C_VEL
LIN {X 0,Y 481.609,Z 143.495,A -85,B 0,C 180,E1 -6796.855,E2 -6796.855} C_VEL
LIN {X 0,Y 481.649,Z 143.484,A -85,B 0,C 180,E1 -6800.057,E2 -6800.057} C_VEL
LIN {X 0,Y 481.602,Z 143.492,A -85,B 0,C 180,E1 -6803.379,E2 -6803.379} C_VEL
LIN {X 0,Y 481.664,Z 143.484,A -85,B 0,C 180,E1 -6806.327,E2 -6806.327} C_VEL
LIN {X 0,Y 481.626,Z 143.488,A -85,B 0,C 180,E1 -6809.421,E2 -6809.421} C_VEL
LIN {X 0,Y 481.64,Z 143.487,A -85,B 0,C 180,E1 -6812.165,E2 -6812.165} C_VEL
LIN {X 0,Y 481.666,Z 143.486,A -85,B 0,C 180,E1 -6814.967,E2 -6814.967} C_VEL
LIN {X 0,Y 481.629,Z 143.487,A -85,B 0,C 180,E1 -6817.704,E2 -6817.704} C_VEL
LIN {X 0,Y 481.684,Z 143.486,A -85,B 0,C 180,E1 -6820.393,E2 -6820.393} C_VEL
LIN {X 0,Y 481.611,Z 143.49,A -85,B 0,C 180,E1 -6823.031,E2 -6823.031} C_VEL
LIN {X 0,Y 481.665,Z 143.482,A -85,B 0,C 180,E1 -6825.638,E2 -6825.638} C_VEL
LIN {X 0,Y 481.728,Z 143.481,A -85,B 0,C 180,E1 -6828.215,E2 -6828.215} C_VEL
LIN {X 0,Y 481.705,Z 143.478,A -85,B 0,C 180,E1 -6831.611,E2 -6831.611} C_VEL
LIN {X 0,Y 481.765,Z 143.477,A -85,B 0,C 180,E1 -6834.139,E2 -6834.139} C_VEL
LIN {X 0,Y 481.9,Z 143.454,A -85,B 0,C 180,E1 -6837.493,E2 -6837.493} C_VEL
LIN {X 0,Y 481.903,Z 143.46,A -85,B 0,C 180,E1 -6840,E2 -6840} C_VEL
LIN {X 0,Y 481.9,Z 143.455,A -85,B 0,C 180,E1 -6842.508,E2 -6842.508} C_VEL
LIN {X 0,Y 481.765,Z 143.477,A -85,B 0,C 180,E1 -6845.861,E2 -6845.861} C_VEL
LIN {X 0,Y 481.709,Z 143.479,A -85,B 0,C 180,E1 -6848.39,E2 -6848.39} C_VEL
LIN {X 0,Y 481.73,Z 143.482,A -85,B 0,C 180,E1 -6851.786,E2 -6851.786} C_VEL
LIN {X 0,Y 481.723,Z 143.477,A -85,B 0,C 180,E1 -6855.225,E2 -6855.225} C_VEL
LIN {X 0,Y 481.644,Z 143.485,A -85,B 0,C 180,E1 -6858.725,E2 -6858.725} C_VEL
LIN {X 0,Y 481.624,Z 143.493,A -85,B 0,C 180,E1 -6861.396,E2 -6861.396} C_VEL
LIN {X 0,Y 481.64,Z 143.486,A -85,B 0,C 180,E1 -6864.115,E2 -6864.115} C_VEL
LIN {X 0,Y 481.646,Z 143.488,A -85,B 0,C 180,E1 -6867.117,E2 -6867.117} C_VEL
LIN {X 0,Y 481.595,Z 143.494,A -85,B 0,C 180,E1 -6869.747,E2 -6869.747} C_VEL
LIN {X 0,Y 481.645,Z 143.485,A -85,B 0,C 180,E1 -6872.677,E2 -6872.677} C_VEL
LIN {X 0,Y 481.646,Z 143.492,A -85,B 0,C 180,E1 -6875.202,E2 -6875.202} C_VEL
LIN {X 0,Y 481.627,Z 143.487,A -85,B 0,C 180,E1 -6878.004,E2 -6878.004} C_VEL
LIN {X 0,Y 481.619,Z 143.495,A -85,B 0,C 180,E1 -6881.046,E2 -6881.046} C_VEL
LIN {X 0,Y 481.648,Z 143.486,A -85,B 0,C 180,E1 -6884.459,E2 -6884.459} C_VEL
LIN {X 0,Y 481.61,Z 143.495,A -85,B 0,C 180,E1 -6886.856,E2 -6886.856} C_VEL
LIN {X 0,Y 481.654,Z 143.484,A -85,B 0,C 180,E1 -6890.058,E2 -6890.058} C_VEL
LIN {X 0,Y 481.606,Z 143.491,A -85,B 0,C 180,E1 -6893.38,E2 -6893.38} C_VEL
LIN {X 0,Y 481.67,Z 143.484,A -85,B 0,C 180,E1 -6896.327,E2 -6896.327} C_VEL
LIN {X 0,Y 481.61,Z 143.49,A -85,B 0,C 180,E1 -6899.426,E2 -6899.426} C_VEL
LIN {X 0,Y 481.641,Z 143.489,A -85,B 0,C 180,E1 -6902.165,E2 -6902.165} C_VEL
LIN {X 0,Y 481.646,Z 143.604,A -85,B 0,C 180,E1 -6904.781,E2 -6904.781} C_VEL
LIN {X 0,Y 483.516,Z 153.412,A -85,B 0,C 180,E1 -6906.638,E2 -6906.638} C_VEL
LIN {X 0,Y 483.405,Z 162.386,A -85,B 0,C 180,E1 -6908.228,E2 -6908.228} C_VEL
LIN {X 0,Y 482.653,Z 181.44,A -85,B 0,C 180,E1 -6911.536,E2 -6911.536} C_VEL
LIN {X 0,Y 482.286,Z 193.183,A -85,B 0,C 180,E1 -6913.514,E2 -6913.514} C_VEL
LIN {X 0,Y 484.798,Z 210.069,A -85,B 0,C 180,E1 -6913.863,E2 -6913.863} C_VEL
LIN {X 0,Y 484.141,Z 301.459,A -85,B 0,C 180,E1 -6915.284,E2 -6915.284} C_VEL
LIN {X 0,Y 483.776,Z 315.264,A -85,B 0,C 180,E1 -6915.675,E2 -6915.675} C_VEL
LIN {X 0,Y 483.434,Z 327.145,A -85,B 0,C 180,E1 -6916.175,E2 -6916.175} C_VEL
LIN {X 0,Y 482.932,Z 339.673,A -85,B 0,C 180,E1 -6916.889,E2 -6916.889} C_VEL
LIN {X 0,Y 482.512,Z 350.883,A -85,B 0,C 180,E1 -6917.714,E2 -6917.714} C_VEL
LIN {X 0,Y 482.166,Z 361.107,A -85,B 0,C 180,E1 -6918.652,E2 -6918.652} C_VEL
LIN {X 0,Y 481.722,Z 370.429,A -85,B 0,C 180,E1 -6919.705,E2 -6919.705} C_VEL
LIN {X 0,Y 481.373,Z 379.474,A -85,B 0,C 180,E1 -6920.97,E2 -6920.97} C_VEL
LIN {X 0,Y 481.134,Z 386.758,A -85,B 0,C 180,E1 -6922.235,E2 -6922.235} C_VEL
LIN {X 0,Y 480.944,Z 392.809,A -85,B 0,C 180,E1 -6923.557,E2 -6923.557} C_VEL
LIN {X 0,Y 480.895,Z 397.779,A -85,B 0,C 180,E1 -6924.969,E2 -6924.969} C_VEL
LIN {X 0,Y 480.826,Z 400.094,A -85,B 0,C 180,E1 -6925.809,E2 -6925.809} C_VEL
LIN {X 0,Y 480.888,Z 401.977,A -85,B 0,C 180,E1 -6926.649,E2 -6926.649} C_VEL
LIN {X 0,Y 480.824,Z 403.386,A -85,B 0,C 180,E1 -6927.487,E2 -6927.487} C_VEL
LIN {X 0,Y 480.793,Z 404.388,A -85,B 0,C 180,E1 -6928.325,E2 -6928.325} C_VEL
LIN {X 0,Y 480.762,Z 404.997,A -85,B 0,C 180,E1 -6929.162,E2 -6929.162} C_VEL
LIN {X 0,Y 480.746,Z 405.212,A -85,B 0,C 180,E1 -6930,E2 -6930} C_VEL
LIN {X 0,Y 480.762,Z 404.99,A -85,B 0,C 180,E1 -6930.837,E2 -6930.837} C_VEL
LIN {X 0,Y 480.793,Z 404.372,A -85,B 0,C 180,E1 -6931.675,E2 -6931.675} C_VEL
LIN {X 0,Y 480.824,Z 403.362,A -85,B 0,C 180,E1 -6932.513,E2 -6932.513} C_VEL
LIN {X 0,Y 480.888,Z 401.947,A -85,B 0,C 180,E1 -6933.351,E2 -6933.351} C_VEL
LIN {X 0,Y 480.837,Z 398.972,A -85,B 0,C 180,E1 -6934.611,E2 -6934.611} C_VEL
LIN {X 0,Y 480.916,Z 394.949,A -85,B 0,C 180,E1 -6935.871,E2 -6935.871} C_VEL
LIN {X 0,Y 481.104,Z 388.76,A -85,B 0,C 180,E1 -6937.343,E2 -6937.343} C_VEL
LIN {X 0,Y 481.303,Z 382.001,A -85,B 0,C 180,E1 -6938.608,E2 -6938.608} C_VEL
LIN {X 0,Y 481.619,Z 373.618,A -85,B 0,C 180,E1 -6939.872,E2 -6939.872} C_VEL
LIN {X 0,Y 481.974,Z 364.997,A -85,B 0,C 180,E1 -6940.927,E2 -6940.927} C_VEL
LIN {X 0,Y 482.402,Z 354.485,A -85,B 0,C 180,E1 -6941.971,E2 -6941.971} C_VEL
LIN {X 0,Y 482.751,Z 344.126,A -85,B 0,C 180,E1 -6942.805,E2 -6942.805} C_VEL
LIN {X 0,Y 483.253,Z 332.232,A -85,B 0,C 180,E1 -6943.562,E2 -6943.562} C_VEL
LIN {X 0,Y 483.626,Z 320.198,A -85,B 0,C 180,E1 -6944.141,E2 -6944.141} C_VEL
LIN {X 0,Y 484.001,Z 307.209,A -85,B 0,C 180,E1 -6944.586,E2 -6944.586} C_VEL
LIN {X 0,Y 484.255,Z 293.366,A -85,B 0,C 180,E1 -6944.874,E2 -6944.874} C_VEL
LIN {X 0,Y 484.81,Z 208.748,A -85,B 0,C 180,E1 -6946.18,E2 -6946.18} C_VEL
LIN {X 0,Y 482.244,Z 192.377,A -85,B 0,C 180,E1 -6946.537,E2 -6946.537} C_VEL
LIN {X 0,Y 482.873,Z 173.33,A -85,B 0,C 180,E1 -6949.779,E2 -6949.779} C_VEL
LIN {X 0,Y 483.43,Z 157.933,A -85,B 0,C 180,E1 -6952.433,E2 -6952.433} C_VEL
LIN {X 0,Y 483.334,Z 152.11,A -85,B 0,C 180,E1 -6953.46,E2 -6953.46} C_VEL
LIN {X 0,Y 481.646,Z 143.492,A -85,B 0,C 180,E1 -6955.081,E2 -6955.081} C_VEL
LIN {X 0,Y 481.64,Z 143.493,A -85,B 0,C 180,E1 -6957.835,E2 -6957.835} C_VEL
LIN {X 0,Y 481.608,Z 143.498,A -85,B 0,C 180,E1 -6960.713,E2 -6960.713} C_VEL
LIN {X 0,Y 481.674,Z 143.485,A -85,B 0,C 180,E1 -6963.728,E2 -6963.728} C_VEL
LIN {X 0,Y 481.603,Z 143.495,A -85,B 0,C 180,E1 -6966.748,E2 -6966.748} C_VEL
LIN {X 0,Y 481.652,Z 143.487,A -85,B 0,C 180,E1 -6969.942,E2 -6969.942} C_VEL
LIN {X 0,Y 481.615,Z 143.496,A -85,B 0,C 180,E1 -6973.302,E2 -6973.302} C_VEL
LIN {X 0,Y 481.645,Z 143.487,A -85,B 0,C 180,E1 -6975.641,E2 -6975.641} C_VEL
LIN {X 0,Y 481.618,Z 143.495,A -85,B 0,C 180,E1 -6978.954,E2 -6978.954} C_VEL
LIN {X 0,Y 481.625,Z 143.489,A -85,B 0,C 180,E1 -6981.996,E2 -6981.996} C_VEL
LIN {X 0,Y 481.673,Z 143.483,A -85,B 0,C 180,E1 -6985.316,E2 -6985.316} C_VEL
LIN {X 0,Y 481.621,Z 143.491,A -85,B 0,C 180,E1 -6988.309,E2 -6988.309} C_VEL
LIN {X 0,Y 481.626,Z 143.489,A -85,B 0,C 180,E1 -6991.213,E2 -6991.213} C_VEL
LIN {X 0,Y 481.635,Z 143.485,A -85,B 0,C 180,E1 -6994.039,E2 -6994.039} C_VEL
LIN {X 0,Y 481.645,Z 143.485,A -85,B 0,C 180,E1 -6996.818,E2 -6996.818} C_VEL
LIN {X 0,Y 481.65,Z 143.485,A -85,B 0,C 180,E1 -6999.5,E2 -6999.5} C_VEL
LIN {X 0,Y 481.645,Z 143.488,A -85,B 0,C 180,E1 -7002.156,E2 -7002.156} C_VEL
LIN {X 0,Y 481.721,Z 143.476,A -85,B 0,C 180,E1 -7004.775,E2 -7004.775} C_VEL
LIN {X 0,Y 481.727,Z 143.479,A -85,B 0,C 180,E1 -7008.214,E2 -7008.214} C_VEL
LIN {X 0,Y 481.707,Z 143.479,A -85,B 0,C 180,E1 -7011.61,E2 -7011.61} C_VEL
LIN {X 0,Y 481.763,Z 143.476,A -85,B 0,C 180,E1 -7014.139,E2 -7014.139} C_VEL
LIN {X 0,Y 481.898,Z 143.456,A -85,B 0,C 180,E1 -7017.492,E2 -7017.492} C_VEL
LIN {X 0,Y 481.901,Z 143.459,A -85,B 0,C 180,E1 -7020,E2 -7020} C_VEL
LIN {X 0,Y 481.898,Z 143.455,A -85,B 0,C 180,E1 -7022.507,E2 -7022.507} C_VEL
LIN {X 0,Y 481.763,Z 143.477,A -85,B 0,C 180,E1 -7025.861,E2 -7025.861} C_VEL
LIN {X 0,Y 481.706,Z 143.481,A -85,B 0,C 180,E1 -7028.389,E2 -7028.389} C_VEL
LIN {X 0,Y 481.726,Z 143.486,A -85,B 0,C 180,E1 -7031.785,E2 -7031.785} C_VEL
LIN {X 0,Y 481.72,Z 143.484,A -85,B 0,C 180,E1 -7035.225,E2 -7035.225} C_VEL
LIN {X 0,Y 481.695,Z 143.482,A -85,B 0,C 180,E1 -7038.722,E2 -7038.722} C_VEL
LIN {X 0,Y 481.633,Z 143.495,A -85,B 0,C 180,E1 -7041.395,E2 -7041.395} C_VEL
LIN {X 0,Y 481.678,Z 143.55,A -85,B 0,C 180,E1 -7042.746,E2 -7042.746} C_VEL
LIN {X 0,Y 482.812,Z 150.019,A -85,B 0,C 180,E1 -7044.052,E2 -7044.052} C_VEL
LIN {X 0,Y 482.488,Z 165.814,A -85,B 0,C 180,E1 -7047.073,E2 -7047.073} C_VEL
LIN {X 0,Y 482.408,Z 168.17,A -85,B 0,C 180,E1 -7047.521,E2 -7047.521} C_VEL
LIN {X 0,Y 485.001,Z 182.003,A -85,B 0,C 180,E1 -7047.845,E2 -7047.845} C_VEL
LIN {X 0,Y 484.21,Z 276.319,A -85,B 0,C 180,E1 -7049.326,E2 -7049.326} C_VEL
LIN {X 0,Y 483.9,Z 289.629,A -85,B 0,C 180,E1 -7049.71,E2 -7049.71} C_VEL
LIN {X 0,Y 483.609,Z 302.605,A -85,B 0,C 180,E1 -7050.271,E2 -7050.271} C_VEL
LIN {X 0,Y 483.212,Z 314.791,A -85,B 0,C 180,E1 -7050.988,E2 -7050.988} C_VEL
LIN {X 0,Y 482.744,Z 326.194,A -85,B 0,C 180,E1 -7051.847,E2 -7051.847} C_VEL
LIN {X 0,Y 482.28,Z 336.951,A -85,B 0,C 180,E1 -7052.876,E2 -7052.876} C_VEL
LIN {X 0,Y 481.904,Z 346.138,A -85,B 0,C 180,E1 -7053.963,E2 -7053.963} C_VEL
LIN {X 0,Y 481.56,Z 354.56,A -85,B 0,C 180,E1 -7055.188,E2 -7055.188} C_VEL
LIN {X 0,Y 481.251,Z 362.056,A -85,B 0,C 180,E1 -7056.565,E2 -7056.565} C_VEL
LIN {X 0,Y 481.079,Z 367.862,A -85,B 0,C 180,E1 -7057.921,E2 -7057.921} C_VEL
LIN {X 0,Y 480.919,Z 372.215,A -85,B 0,C 180,E1 -7059.239,E2 -7059.239} C_VEL
LIN {X 0,Y 480.829,Z 375.356,A -85,B 0,C 180,E1 -7060.532,E2 -7060.532} C_VEL
LIN {X 0,Y 480.765,Z 377.43,A -85,B 0,C 180,E1 -7061.796,E2 -7061.796} C_VEL
LIN {X 0,Y 480.692,Z 378.757,A -85,B 0,C 180,E1 -7063.406,E2 -7063.406} C_VEL
LIN {X 0,Y 480.76,Z 378.767,A -85,B 0,C 180,E1 -7064.562,E2 -7064.562} C_VEL
LIN {X 0,Y 480.765,Z 377.996,A -85,B 0,C 180,E1 -7065.749,E2 -7065.749} C_VEL
LIN {X 0,Y 480.782,Z 376.384,A -85,B 0,C 180,E1 -7066.961,E2 -7066.961} C_VEL
LIN {X 0,Y 480.853,Z 373.852,A -85,B 0,C 180,E1 -7068.193,E2 -7068.193} C_VEL
LIN {X 0,Y 480.998,Z 369.641,A -85,B 0,C 180,E1 -7069.633,E2 -7069.633} C_VEL
LIN {X 0,Y 480.399,Z 367.366,A -85,B 0,C 180,E1 -7070.279,E2 -7070.279} C_VEL
LIN {X 0,Y 477.677,Z 363.278,A -85,B 0,C 180,E1 -7071.312,E2 -7071.312} C_VEL
LIN {X 0,Y 474.993,Z 358.559,A -85,B 0,C 180,E1 -7072.314,E2 -7072.314} C_VEL
LIN {X 0,Y 474.456,Z 355.246,A -85,B 0,C 180,E1 -7072.903,E2 -7072.903} C_VEL
LIN {X 0,Y 474.778,Z 347.228,A -85,B 0,C 180,E1 -7074.114,E2 -7074.114} C_VEL
LIN {X 0,Y 475.288,Z 337.44,A -85,B 0,C 180,E1 -7075.3,E2 -7075.3} C_VEL
LIN {X 0,Y 475.73,Z 326.6,A -85,B 0,C 180,E1 -7076.36,E2 -7076.36} C_VEL
LIN {X 0,Y 476.187,Z 315.244,A -85,B 0,C 180,E1 -7077.234,E2 -7077.234} C_VEL
LIN {X 0,Y 476.587,Z 303.616,A -85,B 0,C 180,E1 -7077.936,E2 -7077.936} C_VEL
LIN {X 0,Y 476.971,Z 291.811,A -85,B 0,C 180,E1 -7078.476,E2 -7078.476} C_VEL
LIN {X 0,Y 477.165,Z 278.61,A -85,B 0,C 180,E1 -7078.895,E2 -7078.895} C_VEL
LIN {X 0,Y 477.407,Z 260.572,A -85,B 0,C 180,E1 -7079.217,E2 -7079.217} C_VEL
LIN {X 0,Y 478.056,Z 182.397,A -85,B 0,C 180,E1 -7080.435,E2 -7080.435} C_VEL
LIN {X 0,Y 475.376,Z 168.194,A -85,B 0,C 180,E1 -7080.769,E2 -7080.769} C_VEL
LIN {X 0,Y 475.944,Z 153.715,A -85,B 0,C 180,E1 -7083.706,E2 -7083.706} C_VEL
LIN {X 0,Y 475.556,Z 149.354,A -85,B 0,C 180,E1 -7084.623,E2 -7084.623} C_VEL
LIN {X 0,Y 474.607,Z 144.367,A -85,B 0,C 180,E1 -7085.738,E2 -7085.738} C_VEL
LIN {X 0,Y 474.651,Z 144.359,A -85,B 0,C 180,E1 -7089.185,E2 -7089.185} C_VEL
LIN {X 0,Y 474.627,Z 144.36,A -85,B 0,C 180,E1 -7091.884,E2 -7091.884} C_VEL
LIN {X 0,Y 474.683,Z 144.359,A -85,B 0,C 180,E1 -7094.544,E2 -7094.544} C_VEL
LIN {X 0,Y 474.689,Z 144.355,A -85,B 0,C 180,E1 -7098.038,E2 -7098.038} C_VEL
LIN {X 0,Y 474.66,Z 144.355,A -85,B 0,C 180,E1 -7101.486,E2 -7101.486} C_VEL
LIN {X 0,Y 474.731,Z 144.352,A -85,B 0,C 180,E1 -7104.052,E2 -7104.052} C_VEL
LIN {X 0,Y 474.868,Z 144.33,A -85,B 0,C 180,E1 -7107.455,E2 -7107.455} C_VEL
LIN {X 0,Y 474.876,Z 144.335,A -85,B 0,C 180,E1 -7110,E2 -7110} C_VEL
LIN {X 0,Y 474.867,Z 144.331,A -85,B 0,C 180,E1 -7112.545,E2 -7112.545} C_VEL
LIN {X 0,Y 474.731,Z 144.354,A -85,B 0,C 180,E1 -7115.948,E2 -7115.948} C_VEL
LIN {X 0,Y 474.661,Z 144.356,A -85,B 0,C 180,E1 -7118.515,E2 -7118.515} C_VEL
LIN {X 0,Y 474.689,Z 144.357,A -85,B 0,C 180,E1 -7121.963,E2 -7121.963} C_VEL
LIN {X 0,Y 474.684,Z 144.356,A -85,B 0,C 180,E1 -7125.456,E2 -7125.456} C_VEL
LIN {X 0,Y 474.599,Z 144.363,A -85,B 0,C 180,E1 -7129.013,E2 -7129.013} C_VEL
LIN {X 0,Y 474.57,Z 144.372,A -85,B 0,C 180,E1 -7131.73,E2 -7131.73} C_VEL
LIN {X 0,Y 474.62,Z 144.36,A -85,B 0,C 180,E1 -7134.495,E2 -7134.495} C_VEL
LIN {X 0,Y 474.592,Z 144.369,A -85,B 0,C 180,E1 -7137.326,E2 -7137.326} C_VEL
LIN {X 0,Y 474.552,Z 144.368,A -85,B 0,C 180,E1 -7140.234,E2 -7140.234} C_VEL
LIN {X 0,Y 474.609,Z 144.368,A -85,B 0,C 180,E1 -7143.222,E2 -7143.222} C_VEL
LIN {X 0,Y 474.576,Z 144.365,A -85,B 0,C 180,E1 -7146.324,E2 -7146.324} C_VEL
LIN {X 0,Y 474.595,Z 144.365,A -85,B 0,C 180,E1 -7149.643,E2 -7149.643} C_VEL
LIN {X 0,Y 474.563,Z 144.372,A -85,B 0,C 180,E1 -7152.939,E2 -7152.939} C_VEL
LIN {X 0,Y 474.595,Z 144.363,A -85,B 0,C 180,E1 -7155.894,E2 -7155.894} C_VEL
LIN {X 0,Y 474.584,Z 144.368,A -85,B 0,C 180,E1 -7159.339,E2 -7159.339} C_VEL
LIN {X 0,Y 474.584,Z 144.364,A -85,B 0,C 180,E1 -7161.707,E2 -7161.707} C_VEL
LIN {X 0,Y 474.604,Z 144.368,A -85,B 0,C 180,E1 -7164.724,E2 -7164.724} C_VEL
LIN {X 0,Y 474.619,Z 144.36,A -85,B 0,C 180,E1 -7167.787,E2 -7167.787} C_VEL
LIN {X 0,Y 474.586,Z 144.37,A -85,B 0,C 180,E1 -7170.892,E2 -7170.892} C_VEL
LIN {X 0,Y 474.582,Z 144.364,A -85,B 0,C 180,E1 -7173.624,E2 -7173.624} C_VEL
LIN {X 0,Y 474.591,Z 144.371,A -85,B 0,C 180,E1 -7176.653,E2 -7176.653} C_VEL
LIN {X 0,Y 474.632,Z 144.361,A -85,B 0,C 180,E1 -7180.089,E2 -7180.089} C_VEL
LIN {X 0,Y 474.586,Z 144.368,A -85,B 0,C 180,E1 -7182.772,E2 -7182.772} C_VEL
LIN {X 0,Y 474.624,Z 144.359,A -85,B 0,C 180,E1 -7185.421,E2 -7185.421} C_VEL
LIN {X 0,Y 474.686,Z 144.356,A -85,B 0,C 180,E1 -7188.037,E2 -7188.037} C_VEL
LIN {X 0,Y 474.654,Z 144.356,A -85,B 0,C 180,E1 -7191.486,E2 -7191.486} C_VEL
LIN {X 0,Y 474.728,Z 144.352,A -85,B 0,C 180,E1 -7194.052,E2 -7194.052} C_VEL
LIN {X 0,Y 474.865,Z 144.33,A -85,B 0,C 180,E1 -7197.456,E2 -7197.456} C_VEL
LIN {X 0,Y 474.873,Z 144.336,A -85,B 0,C 180,E1 -7200,E2 -7200} C_VEL
LIN {X 0,Y 474.865,Z 144.331,A -85,B 0,C 180,E1 -7202.545,E2 -7202.545} C_VEL
LIN {X 0,Y 474.728,Z 144.354,A -85,B 0,C 180,E1 -7205.949,E2 -7205.949} C_VEL
LIN {X 0,Y 474.658,Z 144.356,A -85,B 0,C 180,E1 -7208.515,E2 -7208.515} C_VEL
LIN {X 0,Y 474.687,Z 144.357,A -85,B 0,C 180,E1 -7211.963,E2 -7211.963} C_VEL
LIN {X 0,Y 474.682,Z 144.357,A -85,B 0,C 180,E1 -7215.457,E2 -7215.457} C_VEL
LIN {X 0,Y 474.598,Z 144.364,A -85,B 0,C 180,E1 -7219.013,E2 -7219.013} C_VEL
LIN {X 0,Y 474.57,Z 144.372,A -85,B 0,C 180,E1 -7221.73,E2 -7221.73} C_VEL
LIN {X 0,Y 474.62,Z 144.36,A -85,B 0,C 180,E1 -7224.495,E2 -7224.495} C_VEL
LIN {X 0,Y 474.592,Z 144.37,A -85,B 0,C 180,E1 -7227.327,E2 -7227.327} C_VEL
LIN {X 0,Y 474.545,Z 144.369,A -85,B 0,C 180,E1 -7230.235,E2 -7230.235} C_VEL
LIN {X 0,Y 474.61,Z 144.368,A -85,B 0,C 180,E1 -7233.223,E2 -7233.223} C_VEL
LIN {X 0,Y 474.568,Z 144.366,A -85,B 0,C 180,E1 -7236.326,E2 -7236.326} C_VEL
LIN {X 0,Y 474.597,Z 144.365,A -85,B 0,C 180,E1 -7239.644,E2 -7239.644} C_VEL
LIN {X 0,Y 474.572,Z 144.366,A -85,B 0,C 180,E1 -7242.23,E2 -7242.23} C_VEL
LIN {X 0,Y 474.611,Z 144.366,A -85,B 0,C 180,E1 -7245.299,E2 -7245.299} C_VEL
LIN {X 0,Y 474.589,Z 144.364,A -85,B 0,C 180,E1 -7248.212,E2 -7248.212} C_VEL
LIN {X 0,Y 474.616,Z 144.363,A -85,B 0,C 180,E1 -7250.452,E2 -7250.452} C_VEL
LIN {X 0,Y 474.569,Z 144.366,A -85,B 0,C 180,E1 -7253.675,E2 -7253.675} C_VEL
LIN {X 0,Y 474.612,Z 144.369,A -85,B 0,C 180,E1 -7256.778,E2 -7256.778} C_VEL
LIN {X 0,Y 474.549,Z 144.369,A -85,B 0,C 180,E1 -7259.766,E2 -7259.766} C_VEL
LIN {X 0,Y 474.601,Z 144.367,A -85,B 0,C 180,E1 -7262.685,E2 -7262.685} C_VEL
LIN {X 0,Y 474.623,Z 144.499,A -85,B 0,C 180,E1 -7264.591,E2 -7264.591} C_VEL
LIN {X 0,Y 476.555,Z 154.62,A -85,B 0,C 180,E1 -7266.536,E2 -7266.536} C_VEL
LIN {X 0,Y 476.459,Z 163.624,A -85,B 0,C 180,E1 -7268.156,E2 -7268.156} C_VEL
LIN {X 0,Y 475.662,Z 182.483,A -85,B 0,C 180,E1 -7271.478,E2 -7271.478} C_VEL
LIN {X 0,Y 475.291,Z 192.697,A -85,B 0,C 180,E1 -7273.258,E2 -7273.258} C_VEL
LIN {X 0,Y 477.943,Z 210.136,A -85,B 0,C 180,E1 -7273.636,E2 -7273.636} C_VEL
LIN {X 0,Y 477.275,Z 300.776,A -85,B 0,C 180,E1 -7275.067,E2 -7275.067} C_VEL
LIN {X 0,Y 476.92,Z 313.98,A -85,B 0,C 180,E1 -7275.438,E2 -7275.438} C_VEL
LIN {X 0,Y 476.512,Z 326.707,A -85,B 0,C 180,E1 -7275.97,E2 -7275.97} C_VEL
LIN {X 0,Y 476.031,Z 338.839,A -85,B 0,C 180,E1 -7276.663,E2 -7276.663} C_VEL
LIN {X 0,Y 475.535,Z 350.614,A -85,B 0,C 180,E1 -7277.536,E2 -7277.536} C_VEL
LIN {X 0,Y 475.122,Z 360.811,A -85,B 0,C 180,E1 -7278.481,E2 -7278.481} C_VEL
LIN {X 0,Y 474.714,Z 370.165,A -85,B 0,C 180,E1 -7279.551,E2 -7279.551} C_VEL
LIN {X 0,Y 474.332,Z 379.225,A -85,B 0,C 180,E1 -7280.835,E2 -7280.835} C_VEL
LIN {X 0,Y 474.059,Z 386.521,A -85,B 0,C 180,E1 -7282.118,E2 -7282.118} C_VEL
LIN {X 0,Y 473.905,Z 391.448,A -85,B 0,C 180,E1 -7283.186,E2 -7283.186} C_VEL
LIN {X 0,Y 473.84,Z 396.232,A -85,B 0,C 180,E1 -7284.468,E2 -7284.468} C_VEL
LIN {X 0,Y 473.733,Z 399.884,A -85,B 0,C 180,E1 -7285.746,E2 -7285.746} C_VEL
LIN {X 0,Y 473.795,Z 401.772,A -85,B 0,C 180,E1 -7286.598,E2 -7286.598} C_VEL
LIN {X 0,Y 473.742,Z 403.186,A -85,B 0,C 180,E1 -7287.449,E2 -7287.449} C_VEL
LIN {X 0,Y 473.69,Z 404.801,A -85,B 0,C 180,E1 -7289.15,E2 -7289.15} C_VEL
LIN {X 0,Y 473.673,Z 405.018,A -85,B 0,C 180,E1 -7290,E2 -7290} C_VEL
LIN {X 0,Y 473.69,Z 404.798,A -85,B 0,C 180,E1 -7290.85,E2 -7290.85} C_VEL
LIN {X 0,Y 473.742,Z 403.169,A -85,B 0,C 180,E1 -7292.551,E2 -7292.551} C_VEL
LIN {X 0,Y 473.795,Z 401.753,A -85,B 0,C 180,E1 -7293.401,E2 -7293.401} C_VEL
LIN {X 0,Y 473.76,Z 398.776,A -85,B 0,C 180,E1 -7294.68,E2 -7294.68} C_VEL
LIN {X 0,Y 473.824,Z 394.751,A -85,B 0,C 180,E1 -7295.959,E2 -7295.959} C_VEL
LIN {X 0,Y 474.014,Z 388.559,A -85,B 0,C 180,E1 -7297.454,E2 -7297.454} C_VEL
LIN {X 0,Y 474.261,Z 381.802,A -85,B 0,C 180,E1 -7298.736,E2 -7298.736} C_VEL
LIN {X 0,Y 474.559,Z 373.418,A -85,B 0,C 180,E1 -7300.021,E2 -7300.021} C_VEL
LIN {X 0,Y 474.968,Z 364.798,A -85,B 0,C 180,E1 -7301.09,E2 -7301.09} C_VEL
LIN {X 0,Y 475.419,Z 354.495,A -85,B 0,C 180,E1 -7302.13,E2 -7302.13} C_VEL
LIN {X 0,Y 475.806,Z 343.922,A -85,B 0,C 180,E1 -7302.996,E2 -7302.996} C_VEL
LIN {X 0,Y 476.354,Z 332.031,A -85,B 0,C 180,E1 -7303.762,E2 -7303.762} C_VEL
LIN {X 0,Y 476.744,Z 320.013,A -85,B 0,C 180,E1 -7304.35,E2 -7304.35} C_VEL
LIN {X 0,Y 477.14,Z 307.053,A -85,B 0,C 180,E1 -7304.801,E2 -7304.801} C_VEL
LIN {X 0,Y 477.404,Z 293.307,A -85,B 0,C 180,E1 -7305.092,E2 -7305.092} C_VEL
LIN {X 0,Y 477.964,Z 209.456,A -85,B 0,C 180,E1 -7306.411,E2 -7306.411} C_VEL
LIN {X 0,Y 475.285,Z 192.056,A -85,B 0,C 180,E1 -7306.816,E2 -7306.816} C_VEL
LIN {X 0,Y 475.986,Z 173.19,A -85,B 0,C 180,E1 -7310.077,E2 -7310.077} C_VEL
LIN {X 0,Y 476.646,Z 156.49,A -85,B 0,C 180,E1 -7313,E2 -7313} C_VEL
LIN {X 0,Y 475.895,Z 150.899,A -85,B 0,C 180,E1 -7314.038,E2 -7314.038} C_VEL
LIN {X 0,Y 474.624,Z 144.367,A -85,B 0,C 180,E1 -7315.314,E2 -7315.314} C_VEL
LIN {X 0,Y 474.587,Z 144.369,A -85,B 0,C 180,E1 -7318.286,E2 -7318.286} C_VEL
LIN {X 0,Y 474.573,Z 144.377,A -85,B 0,C 180,E1 -7321.219,E2 -7321.219} C_VEL
LIN {X 0,Y 474.615,Z 144.362,A -85,B 0,C 180,E1 -7324.242,E2 -7324.242} C_VEL
LIN {X 0,Y 474.538,Z 144.378,A -85,B 0,C 180,E1 -7327.388,E2 -7327.388} C_VEL
LIN {X 0,Y 474.597,Z 144.368,A -85,B 0,C 180,E1 -7329.643,E2 -7329.643} C_VEL
LIN {X 0,Y 474.566,Z 144.374,A -85,B 0,C 180,E1 -7332.939,E2 -7332.939} C_VEL
LIN {X 0,Y 474.576,Z 144.367,A -85,B 0,C 180,E1 -7335.891,E2 -7335.891} C_VEL
LIN {X 0,Y 474.594,Z 144.369,A -85,B 0,C 180,E1 -7339.044,E2 -7339.044} C_VEL
LIN {X 0,Y 474.585,Z 144.365,A -85,B 0,C 180,E1 -7341.707,E2 -7341.707} C_VEL
LIN {X 0,Y 474.606,Z 144.368,A -85,B 0,C 180,E1 -7344.724,E2 -7344.724} C_VEL
LIN {X 0,Y 474.616,Z 144.36,A -85,B 0,C 180,E1 -7347.786,E2 -7347.786} C_VEL
LIN {X 0,Y 474.569,Z 144.371,A -85,B 0,C 180,E1 -7350.895,E2 -7350.895} C_VEL
LIN {X 0,Y 474.582,Z 144.361,A -85,B 0,C 180,E1 -7353.623,E2 -7353.623} C_VEL
LIN {X 0,Y 474.591,Z 144.365,A -85,B 0,C 180,E1 -7356.652,E2 -7356.652} C_VEL
LIN {X 0,Y 474.604,Z 144.367,A -85,B 0,C 180,E1 -7360.087,E2 -7360.087} C_VEL
LIN {X 0,Y 474.581,Z 144.368,A -85,B 0,C 180,E1 -7362.772,E2 -7362.772} C_VEL
LIN {X 0,Y 474.62,Z 144.358,A -85,B 0,C 180,E1 -7365.42,E2 -7365.42} C_VEL
LIN {X 0,Y 474.685,Z 144.356,A -85,B 0,C 180,E1 -7368.037,E2 -7368.037} C_VEL
LIN {X 0,Y 474.656,Z 144.356,A -85,B 0,C 180,E1 -7371.485,E2 -7371.485} C_VEL
LIN {X 0,Y 474.726,Z 144.353,A -85,B 0,C 180,E1 -7374.051,E2 -7374.051} C_VEL
LIN {X 0,Y 474.863,Z 144.333,A -85,B 0,C 180,E1 -7377.455,E2 -7377.455} C_VEL
LIN {X 0,Y 474.871,Z 144.335,A -85,B 0,C 180,E1 -7380,E2 -7380} C_VEL
LIN {X 0,Y 474.863,Z 144.332,A -85,B 0,C 180,E1 -7382.544,E2 -7382.544} C_VEL
LIN {X 0,Y 474.726,Z 144.353,A -85,B 0,C 180,E1 -7385.948,E2 -7385.948} C_VEL
LIN {X 0,Y 474.655,Z 144.359,A -85,B 0,C 180,E1 -7388.514,E2 -7388.514} C_VEL
LIN {X 0,Y 474.684,Z 144.361,A -85,B 0,C 180,E1 -7391.963,E2 -7391.963} C_VEL
LIN {X 0,Y 474.679,Z 144.363,A -85,B 0,C 180,E1 -7395.456,E2 -7395.456} C_VEL
LIN {X 0,Y 474.649,Z 144.361,A -85,B 0,C 180,E1 -7399.011,E2 -7399.011} C_VEL
LIN {X 0,Y 474.576,Z 144.374,A -85,B 0,C 180,E1 -7401.729,E2 -7401.729} C_VEL
LIN {X 0,Y 474.639,Z 144.569,A -85,B 0,C 180,E1 -7402.585,E2 -7402.585} C_VEL
LIN {X 0,Y 475.862,Z 151.309,A -85,B 0,C 180,E1 -7403.962,E2 -7403.962} C_VEL
LIN {X 0,Y 475.516,Z 167.766,A -85,B 0,C 180,E1 -7407.15,E2 -7407.15} C_VEL
LIN {X 0,Y 475.485,Z 168.431,A -85,B 0,C 180,E1 -7407.271,E2 -7407.271} C_VEL
LIN {X 0,Y 478.213,Z 182.651,A -85,B 0,C 180,E1 -7407.607,E2 -7407.607} C_VEL
LIN {X 0,Y 477.363,Z 275.786,A -85,B 0,C 180,E1 -7409.09,E2 -7409.09} C_VEL
LIN {X 0,Y 477.057,Z 289.566,A -85,B 0,C 180,E1 -7409.488,E2 -7409.488} C_VEL
LIN {X 0,Y 476.758,Z 301.764,A -85,B 0,C 180,E1 -7410.013,E2 -7410.013} C_VEL
LIN {X 0,Y 476.322,Z 313.943,A -85,B 0,C 180,E1 -7410.722,E2 -7410.722} C_VEL
LIN {X 0,Y 475.828,Z 325.879,A -85,B 0,C 180,E1 -7411.623,E2 -7411.623} C_VEL
LIN {X 0,Y 475.323,Z 336.619,A -85,B 0,C 180,E1 -7412.65,E2 -7412.65} C_VEL
LIN {X 0,Y 474.902,Z 346.704,A -85,B 0,C 180,E1 -7413.86,E2 -7413.86} C_VEL
LIN {X 0,Y 474.529,Z 354.565,A -85,B 0,C 180,E1 -7415.023,E2 -7415.023} C_VEL
LIN {X 0,Y 474.229,Z 361.803,A -85,B 0,C 180,E1 -7416.355,E2 -7416.355} C_VEL
LIN {X 0,Y 474.033,Z 368.007,A -85,B 0,C 180,E1 -7417.813,E2 -7417.813} C_VEL
